{attribute 'monitoring':='call'}
//List of movers managed by this station
PROPERTY AssignedMovers : I_CH_List
GET
AssignedMovers := THIS^.fbAssignedMovers;
END_GET
END_PROPERTY

METHOD DeleteMoversQueue : HRESULT
VAR
	ipTempMover : I_XP_Mover;
END_VAR
//Not allowed in enabled state
IF THIS^.ipXPSystem.Enabled THEN
	DeleteMoversQueue := E_FAIL;
	RETURN;
END_IF


//Delete intormation in linked mover
THIS^.fbAssignedMovers.ResetIterator();
WHILE THIS^.fbAssignedMovers.HasNextObject() DO
	IF ToXPMover(THIS^.fbAssignedMovers.GetNextObject(),ipTempMover) THEN
		ipTempMover.ParentStation := 0;
	END_IF	
END_WHILE

//Clear list
fbAssignedMovers.Clear();

DeleteMoversQueue := S_OK;
END_METHOD

METHOD FB_exit : BOOL
VAR_INPUT
	bInCopyCode : BOOL; // if TRUE, the exit method is called for exiting an instance that is copied afterwards (online change).
END_VAR
VAR
	pFbPath : POINTER TO FB_XP_Path;
	ipObject : I_CH_Object;
	ipPath : I_XP_Path;
END_VAR
//Clear list, delete dynamic_creation path objects
WHILE NOT THIS^.fbListPathAhead.IsEmpty DO
	ipObject := fbListPathAhead.GetRandomObject();
	fbListPathAhead.RemoveObject(ipObject);
	
	__QUERYINTERFACE(ipObject, ipPath) ;
	pFbPath := ipPath.PointerToThis;
	__DELETE(pFbPath);
END_WHILE
END_METHOD

METHOD FB_init : BOOL
VAR_INPUT
	bInitRetains : BOOL; // if TRUE, the retain variables are initialized (warm start / cold start)
	bInCopyCode : BOOL;  // if TRUE, the instance afterwards gets moved into the copy code (online change)
	
	ipSystem 			: I_CH_Object;
	ipAccocietedTrack 	: I_XP_Track;//track on which the station is located
	sUniqueName			: STRING;		//expl.:'Loading' unique identification for this station
	sTargetGroup		: STRING;	//to which group of stations does this station belong? e.g. several stations can belong to one 'Infeed' if this is implemented redundantly.
	nMoverQueueSize 	: UINT;
	xPos				: LREAL; 	
	yPos				: LREAL; 	
END_VAR

VAR_INST
	{attribute 'hide'}
	bFBInitCalledOnce : BOOL; //Do the following code once during start up and not during onlinechange
END_VAR

VAR 



END_VAR
//Do the following code once during start up and not during onlinechange
IF NOT bFBInitCalledOnce THEN 
	
	(* Register to the Xplanar System
	   1. Test if the interface exists
	   2. Test if the object implements a "System for Mover" interface 
	*)
	IF ipSystem <> 0 AND_THEN __QUERYINTERFACE(ipSystem,THIS^.ipXpSystem) THEN
		THIS^.ipXpSystem.RegisterStation(THIS^);
	ELSE
		bErrorDuringFbInit := TRUE;
	END_IF

	
	// 0 = get closest track (in step configure)
	IF ipAccocietedTrack <> 0 THEN
		THIS^.ipAccocietedTrack := ipAccocietedTrack;
		bTrackIsSetInFbInit := TRUE;
	END_IF
	 
	
	//"" is maybe entered in an waiting or dynamic station and the name is not important
	IF sUniqueName <> '' THEN 
		THIS^.fbSourceInfo.sName := sUniqueName;
	ELSE
		sUniqueName := THIS^.fbSourceInfo.sName;
	END_IF

	
	//"" is maybe entered in an waiting or dynamic station and the name is not important
	IF sTargetGroup <> '' THEN 
		THIS^.sTargetGroup := sTargetGroup;
	ELSE
		THIS^.sTargetGroup := THIS^.fbSourceInfo.sName;
	END_IF

	
	THIS^.nMoverQueueSize 		:= nMoverQueueSize;
	THIS^.fbPositionPlanned.x 	:= xPos;
	THIS^.fbPositionPlanned.y 	:= yPos;


	THIS^.fbTrigger.FB_init(FALSE,FALSE, THIS^.ipXpSystem);

END_IF

bFBInitCalledOnce := TRUE;
END_METHOD

{attribute 'monitoring':='call'}
PROPERTY Feedback : I_CH_Feedback
GET
Feedback := THIS^.fbFeedback;
END_GET
END_PROPERTY

{attribute 'monitoring':='call'}
//Filter content, movers with one of these targets may not approach or drive over the station
PROPERTY Filter : STRING
GET
Filter := sFilter;
END_GET
SET
sFilter := Filter;
END_SET
END_PROPERTY

(*THIS METHOD uses the A* algorithm TO find the shortest route TO the destination in the network. Returns an INTERFACE with information about the destination found, such as station, path TO destination, path length.
If an interface=0 is returned, then no path can be found at the current time.*)
METHOD GetPathToTarged : I_PathAStarNode
VAR_INPUT
	sTargedStation : REFERENCE TO STRING; //unique station name or group of stations. EmptyString=Any
END_VAR
VAR	
	nDifZero : INT;	///zzz remove

	nIdx : UDINT;
	bCorrectLUID: BOOL;
	bCorrectGroupe : BOOL;
	bFilterBlockThisMover : BOOL;
	bStationIsBlocked : BOOL;
	bDummyStation : BOOL; //Station without movers only to change the dynamics of passing movers;
	bTargedFound : BOOL;
	bImTheAsker : BOOL; // Do not return this station as a targed

	ipActiveStationAStar : I_PathAStarNode;
	ipEmptyPathObj : I_PathAStarNode;
	ipEachPathAhead : I_XP_Path;
	ipPathFoundInOpenList : I_PathAStarNode;
	ipEachAStarNode : I_PathAStarNode;
	ipBesStationAStar : I_PathAStarNode;	
	ipThisStation : I_XP_Station := THIS^;
	
	fPathLength : LREAL;
END_VAR
VAR_INST
	fbLastFoundResult : FB_AStarNode;
END_VAR
VAR_STAT
	fbListNotUsedNodes : FB_CH_List; // Use GetNext() to allways get a not used one
	afbPathAStarNodes : ARRAY[0..(CHALET_BaseComponents.BaseParameterlist.MAX_OBJECTS-1)] OF FB_AStarNode;	
	fbListOpen : FB_CH_List; //To check
	fbListClosed : FB_CH_List; //Allready checked	
END_VAR
//only on first call, add nodes to list of not used objects
IF fbListNotUsedNodes.IsEmpty THEN
	FOR nIdx := 0 TO (CHALET_BaseComponents.BaseParameterlist.MAX_OBJECTS-1) DO
		fbListNotUsedNodes.AddObject(afbPathAStarNodes[nIdx]);
	END_FOR
END_IF

//Clear list
fbListOpen.Clear();
fbListClosed.Clear();

//Init objects in list
fbListNotUsedNodes.ResetIterator();
WHILE fbListNotUsedNodes.HasNextObject() DO
	IF __QUERYINTERFACE(fbListNotUsedNodes.GetNextObject(), ipEachAStarNode) THEN
		IF 	ipEachAStarNode.Station = 0 THEN
			EXIT;//Last used element found, abort
		END_IF
	
		ipEachAStarNode.Station := 0;
		ipEachAStarNode.RouteUsedToNode.Clear();
	END_IF
END_WHILE

//Reset last found result
fbLastFoundResult.Station := 0;
fbLastFoundResult.RouteUsedToNode.Clear();

// Reset once - Use GetNext() to allways get a not used one
fbListNotUsedNodes.ResetIterator();

//This is the start of the search operation. Add this station
__QUERYINTERFACE(fbListNotUsedNodes.GetNextObject(), ipEmptyPathObj);
ipEmptyPathObj.Station := (THIS^);
fbListOpen.AddObject(ipEmptyPathObj);

WHILE NOT fbListOpen.IsEmpty DO
	//Get objet from list with smallest distanse to start-station

	__QUERYINTERFACE(fbListOpen.GetObjectWithLowestNumber(), ipActiveStationAStar);
	//Move objet from open to closed list
	fbListOpen.RemoveObject(ipActiveStationAStar);
	fbListClosed.AddObject(ipActiveStationAStar);
	
	IF ipActiveStationAStar = 0 THEN
		//zzz todo error, this should never happen
		nDifZero := nDifZero / nDifZero;
		CONTINUE;
	END_IF
	
	IF ipBesStationAStar <> 0 AND_THEN ipActiveStationAStar.PathLength > ipBesStationAStar.PathLength THEN
		// if a valid station is allreadyx known, skip all station who allready have a larger distance
		CONTINUE;
	END_IF
	
	bImTheAsker := ipActiveStationAStar.Station = ipThisStation;
	bCorrectLUID := (ipActiveStationAStar.Station.LUID = sTargedStation);
 	bCorrectGroupe := (ipActiveStationAStar.Station.TargetGroupe = sTargedStation) OR (sTargedStation =  XPlanarParameterlist.S_ANY_STATION_NAME);
	bDummyStation := (ipActiveStationAStar.Station.MoverQueueSize = 0);//Station without movers only to change the dynamics of passing movers;
	bFilterBlockThisMover := (ipActiveStationAStar.Station.Filter <>  XPlanarParameterlist.S_ANY_STATION_NAME) AND (ipActiveStationAStar.Station.Filter <> sTargedStation) AND NOT bCorrectLUID; // Correct LUID is stronger than filter
	bStationIsBlocked := (ipActiveStationAStar.Station.CtsEmptySpaceInQueue <= 0 AND NOT bDummyStation) OR NOT ipActiveStationAStar.Station.ReadyToRecvMovers;

	IF (bFilterBlockThisMover OR bStationIsBlocked) AND NOT bImTheAsker THEN
		//Skip
		CONTINUE;
	END_IF
	
	
	IF (bCorrectLUID OR bCorrectGroupe) AND NOT bImTheAsker AND NOT bDummyStation THEN
		//FOUND! - check if way is shorter
		IF ipBesStationAStar=0 OR_ELSE  ipActiveStationAStar.PathLength <= ipBesStationAStar.PathLength THEN
			//shorter - store
			ipBesStationAStar := ipActiveStationAStar;
		END_IF
		
	ELSE		
		// If the destination has not yet been found, set the successor nodes of the current node to the open list
		ipActiveStationAStar.Station.PathsAhead.ResetIterator();
		WHILE ipActiveStationAStar.Station.PathsAhead.HasNextObject() DO
			__QUERYINTERFACE(ipActiveStationAStar.Station.PathsAhead.GetNextObject(), ipEachPathAhead); 
			
			IF fbListClosed.LUIDInList(ipEachPathAhead.StationDestination.LUID) THEN
				// if the successor node is already on the closed list - do nothing, repeate WHILE loop
				CONTINUE;
			END_IF
			
			//Calculate distance to start oh the new found station
			fPathLength := ipActiveStationAStar.PathLength + ipEachPathAhead.Length;
		
			//Check if this station is allready existin in open list - compare if this one is shorter
			IF __QUERYINTERFACE( fbListOpen.FindLUID(ipEachPathAhead.StationDestination.LUID), ipPathFoundInOpenList)  THEN
				IF ipPathFoundInOpenList.PathLength <= fPathLength  THEN
					//object in open list is shorter - do nothing, repeate WHILE loop
					CONTINUE;
				ELSE
					//new object is shorter - remove old object in open lsit
					fbListOpen.RemoveObject(ipPathFoundInOpenList);
				END_IF
			END_IF			
			
			
			//Add this path ahead to open list - set new length
			__QUERYINTERFACE(fbListNotUsedNodes.GetNextObject(), ipEmptyPathObj);
			ipEmptyPathObj.Station := ipEachPathAhead.StationDestination;
			ipEmptyPathObj.RouteUsedToNode.Duplicate(ipActiveStationAStar.RouteUsedToNode);
			ipEmptyPathObj.RouteUsedToNode.AddObject(ipEachPathAhead);
			fbListOpen.AddObject(ipEmptyPathObj);

		END_WHILE
		ipActiveStationAStar.Station.PathsAhead.RestoreIterator();

	END_IF

END_WHILE


//Return station or nothing
IF ipBesStationAStar = 0 THEN
	GetPathToTarged := 0;
ELSE
	//store list in an instance
	fbLastFoundResult.Station := ipBesStationAStar.Station;
	fbLastFoundResult.RouteUsedToNode.Duplicate(ipBesStationAStar.RouteUsedToNode);
	GetPathToTarged := fbLastFoundResult;
END_IF
END_METHOD

METHOD Initialize : HRESULT
VAR
	ipEachStationAhead : I_XP_Station;
	nIdx : UDINT;
END_VAR
VAR_INST
	//This error cannot be reset. Requires a reset cold
	{attribute 'hide'}	
	fbInitError : FB_TcAlarm;
	{attribute 'hide'}	
	fbMissingInterfaceAlarm : FB_TcAlarm;
END_VAR
//Check Error during FB_Init
IF THIS^.bErrorDuringFbInit THEN
	IF NOT fbInitError.bRaised THEN 
		//This error cannot be reset. Requires a reset cold
		fbInitError.CreateEx(stEventEntry:=TC_EVENTS.CHALET_Base_Events.ErrorFBinit, ipSourceInfo := THIS^.fbSourceInfo, bWithConfirmation := FALSE);
		fbInitError.Raise(0);
	END_IF
	Initialize:= E_FAIL;
	THIS^.fbFeedback.HR := Initialize;
	RETURN;
END_IF	

//Interface to System is missing
IF THIS^.ipXpSystem = 0 THEN
	IF NOT fbMissingInterfaceAlarm.bRaised THEN 
		//This error cannot be reset. Requires a reset cold
		fbMissingInterfaceAlarm.CreateEx(stEventEntry:=TC_EVENTS.CHALET_Base_Events.ErrorFBinit, ipSourceInfo := THIS^.fbSourceInfo, bWithConfirmation := FALSE);
		fbMissingInterfaceAlarm.Raise(0);
	END_IF
	Initialize := E_FAIL;
	THIS^.fbFeedback.HR := Initialize;
	RETURN;
END_IF


IF NOT THIS^.bInitDone THEN
	//Busy
	Initialize:= S_PENDING;
	
	//Clean up
	THIS^.DeleteMoversQueue();


	bInitDone := TRUE;
ELSE
	//Done
	Initialize:= S_OK;
END_IF


THIS^.fbFeedback.ActiveCommand 		:= TO_STRING(CHALET_NC.E_NcAxisCommands.Initialize);
THIS^.eActiveCommand 				:= CHALET_NC.E_NcAxisCommands.Initialize;
THIS^.fbFeedback.LastCommandAccepted:= TRUE;	
//Set done or keep in busy state	
THIS^.fbFeedback.HR := Initialize;
END_METHOD

{attribute 'monitoring':='call'}
//[mm] Every mover that leaves or passes the station gets this new gap as a target.
PROPERTY MoverGapAtExit : LREAL
GET
MoverGapAtExit := fMoverGapAtExit;
END_GET
SET
IF MoverGapAtExit < XPlanarParameterlist.F_MOVER_MINIMUM_GAP_ON_TRACK THEN
	MoverGapAtExit := XPlanarParameterlist.F_MOVER_MINIMUM_GAP_ON_TRACK;
END_IF

fMoverGapAtExit := MoverGapAtExit;
END_SET
END_PROPERTY

{attribute 'monitoring':='call'}
//Unique object ID
PROPERTY OID : OTCID
GET
OID := THIS^.fbOptionalTrackUsedInLiveView.MCTOPLC_STD.TrackOID;
END_GET
END_PROPERTY

{attribute 'monitoring':='call'}
//List of paths that lead to stations before this station
PROPERTY PathsAhead : I_CH_List
GET
PathsAhead := THIS^.fbListPathAhead;
END_GET
END_PROPERTY

{attribute 'monitoring':='call'}
//List of paths that lead to stations behind this station
PROPERTY PathsBehinde : I_CH_List
GET
PathsBehinde := THIS^.fbListPathBehind;
END_GET
END_PROPERTY

{attribute 'monitoring':='call'}
//[mm] from the beginning of the assigned track
PROPERTY PositionOnTrack : LREAL
GET
PositionOnTrack := THIS^.fPositionOnTrack;
END_GET
END_PROPERTY

{attribute 'monitoring':='call'}
//Position on the assigned track
PROPERTY PositionOnTrackXY : REFERENCE TO PositionXY
GET
PositionOnTrackXY REF= THIS^.fbPositionOnTrackXY;
END_GET
END_PROPERTY

{attribute 'monitoring':='call'}
//Planned position, not necessarily on the track. Only changeable when the system is disabled
PROPERTY PositionXY : REFERENCE TO  PositionXY
GET
PositionXY REF= THIS^.fbPositionPlanned;
END_GET
END_PROPERTY

(* 
	Use this Methode to calculate time sensitive date once each cycle. Example: read analog input and convert before do get Signal propertie
*)
METHOD PROTECTED Prepare : HRESULT
VAR_INST
	{attribute 'hide'}	
	nLastUpdatedCycleCount : UDINT;
END_VAR

VAR
	nLoopIndex : UINT;
	fExpectedDistanceToParent : LREAL;
	nCycleTime_ms : UDINT;
	bMoverInQueue : BOOL;
	bTempMoverInPosition : BOOL;
	bTempMoverVeloZero : BOOL;
	bTempMoverInMonitoringTime : BOOL;
	bTempMoverThisStationAsTarged : BOOL;
END_VAR
VAR_INST
	{attribute 'hide'}
	nCycleCountInPos : UDINT;
END_VAR
//Check if this Cycle the dates are allready prepared. This is important for time sensitive informations.
IF nLastUpdatedCycleCount <> TwinCAT_SystemInfoVarList._TaskInfo[THIS^.TaskIndex].CycleCount THEN
	nLastUpdatedCycleCount := TwinCAT_SystemInfoVarList._TaskInfo[THIS^.TaskIndex].CycleCount ;


	(* Check if mover is in place. Time and Position window *)
	//If queuesize is zero, mover is never in place.
	IF nMoverQueueSize = 0 OR THIS^.ipAccocietedTrack = 0 OR NOT ipXpSystem.Enabled THEN
		THIS^.bMoversInPlace := FALSE;
		nCycleCountInPos := 0;
	ELSE
		//Get this task cycle Count and time 
		nCycleTime_ms := TwinCAT_SystemInfoVarList._TaskInfo[THIS^.nTaskIndex].CycleTime(*100ns*) / 10_000 ;
		
		bTempMoverInPosition := TRUE; bTempMoverVeloZero := TRUE; bTempMoverThisStationAsTarged := TRUE;
		fExpectedDistanceToParent := 0;
		FOR nLoopIndex := 0 TO (THIS^.nMoverQueueSize-1) DO
			IF THIS^.fbSortedListMoversInQueue.MoversInZone[nLoopIndex] <> 0 THEN
				//Check position and Gap - 1 mover do not have a gap
				IF nLoopIndex <> 0 THEN
					fExpectedDistanceToParent := fExpectedDistanceToParent + THIS^.fbSortedListMoversInQueue.MoversInZone[nLoopIndex].LastCmdTargedGap;
				END_IF
				bMoverInQueue		:= TRUE;
				bTempMoverInPosition := bTempMoverInPosition AND (ABS(THIS^.fbSortedListMoversInQueue.MoversInZone[nLoopIndex].DistToParentStation - fExpectedDistanceToParent) <= fTargetPosWindow );
				bTempMoverVeloZero := bTempMoverVeloZero AND (THIS^.fbSortedListMoversInQueue.MoversInZone[nLoopIndex].PlanarMover.MCTOPLC.SETONTRACK.SetVelo = 0.0);
				bTempMoverThisStationAsTarged := bTempMoverThisStationAsTarged AND ((THIS^.fbSortedListMoversInQueue.MoversInZone[nLoopIndex].TargetStation = THIS^.TargetGroupe) OR (THIS^.fbSortedListMoversInQueue.MoversInZone[nLoopIndex].TargetStation = THIS^.LUID));
			ELSE
				//Missing mover in queue
				bMoverInQueue := FALSE;
				EXIT;
			END_IF
		END_FOR
			
		//start time if mover position is ok
		IF bTempMoverInPosition  THEN
			nCycleCountInPos := nCycleCountInPos + 1;
		ELSE
			nCycleCountInPos := 0;
		END_IF
		
		bTempMoverInMonitoringTime := (UDINT_TO_TIME(nCycleCountInPos * nCycleTime_ms) >= tTargetPosMonitoringTime);
				
		THIS^.bMoversInPlace := bMoverInQueue AND bTempMoverInPosition AND bTempMoverInMonitoringTime AND bTempMoverThisStationAsTarged;// AND bTempMoverVeloZero;
	END_IF
	
	
END_IF
END_METHOD

{attribute 'monitoring':='call'}
//List of stations before this station
PROPERTY StationsAhead : I_CH_List
GET
StationsAhead := THIS^.fbStationsAhead;
END_GET
END_PROPERTY

{attribute 'monitoring':='call'}
//List of stations behinde this station
PROPERTY StationsBehinde : I_CH_List
GET
StationsBehinde := THIS^.fbStationsBehinde;
END_GET
END_PROPERTY

METHOD Update : HRESULT
VAR
	iStation: I_XP_Station;
	bValideStationToStartMove : BOOL;
	ipThisStation : I_XP_Station := THIS^;
	ipPath : I_XP_Path;
	ipRoute : I_CH_List;
	ipMover : I_XP_Mover;
	bValideInterface, bMoverOnSameTrack, bInDecisionDistance : BOOL;
	nIdx : UDINT;
	bStationIsBlocked : BOOL;
END_VAR
//Force to do init befor call update
IF NOT bInitDone THEN
	THIS^.Initialize();
	RETURN;
END_IF

THIS^.Prepare();//Prepare time-critical information, if not already done


// ********************** Set feedback depending on active command *******************************
IF THIS^.eActiveCommand <> E_NcAxisCommands.None THEN
	fbFeedback.ActiveCommand 	:= TO_STRING(THIS^.eActiveCommand);	
END_IF

CASE THIS^.eActiveCommand OF

	E_NcAxisCommands.Initialize:
		fbFeedback.Busy 			:= NOT THIS^.bInitDone;
		fbFeedback.Done 			:= THIS^.bInitDone;
		fbFeedback.ErrorId 			:= 0;
		                        	

	ELSE//External command in subclass
		;
END_CASE


// **********************  Stop to execute commands on .done or .error ***************************
IF fbFeedback.Done OR THIS^.fbFeedback.Error THEN
	eActiveCommand 				:= E_NcAxisCommands.None;
END_IF



// **********************  OnMoverPasses ***************************
// Detect mover who is passing the station and call method for easier overwriting
IF fbTrigger.MoverDetected AND (fbTrigger.MoverAtTrigger <> 0) THEN
	THIS^.OnMoverPasses(fbTrigger.MoverAtTrigger);
END_IF


// **********************  If enabled start station logic ***************************
IF THIS^.ipXpSystem.Enabled THEN
	
	// Process Simulation. 	
	// All functionality packed into one method for easier overwriting
	THIS^.UpdateSimulation();
	
		
	// Interaction with the movers. Sending on to the next station. 
	// All functionality packed into one method for easier overwriting
	THIS^.UpdateMoverInteraction();
	
	
	//The movers have a list of waypoints that they have to travel to on the way to the destination station. 
	//It is checked whether this station is one of these waypoints
	// - if yes, send the mover to the next waypoint and remove this stop from the list
	//Do not wait until mover is at station possition, use fDecisionDistance
	ipXpSystem.Movers.ResetIterator();
	WHILE ipXpSystem.Movers.HasNextObject() DO
		IF __QUERYINTERFACE(ipXpSystem.Movers.GetNextObject(),ipMover) THEN
			ipRoute := ipMover.Route;
			bValideInterface 	:= ipRoute <> 0;
			bMoverOnSameTrack 	:= ipMover.CurrentTrack = ipThisStation.AccocietedTrack;
			bInDecisionDistance := (ABS(ipMover.PositionOnTrack - ipThisStation.PositionOnTrack) < THIS^.fDecisionDistance);
		ELSE 
			bValideInterface := FALSE; bMoverOnSameTrack := FALSE; bInDecisionDistance := FALSE;
		END_IF		
		
		IF bValideInterface AND bMoverOnSameTrack AND bInDecisionDistance THEN
			ipRoute.ResetIterator();
			WHILE ipRoute.HasNextObject() DO
				IF __QUERYINTERFACE(ipRoute.GetNextObject(), ipPath) AND_THEN ipPath.StationStart = ipThisStation THEN
					//Remove this path from route and send to path desination
					ipMover.Route.RemoveObject(ipPath);
					
					//Set new dynamic. Be careful when reducing the deceleration so that the mover can still stop in real time
					IF XPlanarParameterlist.B_STATIONS_OVERRIDE_MOVER_DYN_CONSTRAINT THEN
						ipMover.SetDynConstraint_Path(	V:= THIS^.fMoverVeloAtExit, 
								A:= THIS^.fMoverAccAtExit,
								D:= THIS^.fMoverDecAtExit,
								J:= MC_DEFAULT);
					END_IF

					
					//If mover is standstill in current station, send him away whit the exit gap, else use the in mover stored gap
					IF (ABS(ipMover.PositionOnTrack - THIS^.PositionOnTrack) <= 1.0) THEN
						ipMover.MoveOnTrackToStation(ipStation := ipPath.StationDestination,
													fGap:= THIS^.fMoverGapAtExit);					
					ELSE
						ipMover.MoveOnTrackToStation(ipStation := ipPath.StationDestination,
													fGap:= ipMover.LastCmdTargedGap);
					END_IF	
				END_IF
			END_WHILE
			ipRoute.RestoreIterator();
		END_IF		
	END_WHILE
	ipXpSystem.Movers.RestoreIterator();
	
	
	//Check for errors
	(*The station is blocked. 
	The first mover in the row is correctly positioned in the station. 
	The queue has a size of >1, but now the n+1 mover does not have this station as its destination. 
	However, it cannot overtake. The station never gives the process a ready signal.*)
	IF THIS^.MoverQueueSize > 1 AND THIS^.MoversInQueue[0] <> 0 AND_THEN (THIS^.MoversInQueue[0].TargetStation = THIS^.TargetGroupe OR THIS^.MoversInQueue[0].TargetStation = THIS^.LUID) THEN
		FOR nIdx := 1 TO (CHALET_BaseComponents.BaseParameterlist.MAX_OBJECTS-1) DO
			//Search for Mover with a direrent targed
			IF THIS^.MoversInQueue[nIdx] <> 0 AND_THEN NOT(THIS^.MoversInQueue[nIdx].TargetStation = THIS^.TargetGroupe OR THIS^.MoversInQueue[nIdx].TargetStation = THIS^.LUID) THEN
				//Error
				bStationIsBlocked := TRUE;
				IF NOT fbAlarmStationIsBlocked.bRaised THEN
					//Station is blocked. Mover {0} has {1} as target position but cannot overtake
					fbAlarmStationIsBlocked.CreateEx(TC_Events.CHALET_XPlanar_Events.StationIsBlocked,0,THIS^.fbSourceInfo);
					fbAlarmStationIsBlocked.ipArguments.AddStringByValue(THIS^.MoversInQueue[nIdx].LUID).AddStringByValue(THIS^.MoversInQueue[nIdx].TargetStation);
					fbAlarmStationIsBlocked.Raise(0);
					EXIT;					
				END_IF
			END_IF
		END_FOR
	END_IF
	IF NOT bStationIsBlocked AND fbAlarmStationIsBlocked.bRaised THEN
		fbAlarmStationIsBlocked.Clear(0,0);
	END_IF
	
	
END_IF



// **********************  If disabled clear some bits ***************************
IF NOT THIS^.ipXpSystem.Enabled THEN
	fbAlarmStationIsBlocked.Clear(0,0);
END_IF

Update := S_OK;
END_METHOD

METHOD PROTECTED UpdateMoverInteraction : HRESULT
VAR
	ipFirstMoverInQueue: I_XP_Mover;
	sTargedStation : STRING;
	bMoverValideToSendAway : BOOL;
	bInReachForNewCmd : BOOL;
	bThisStationAsParent : BOOL;
	bFilterDoesNotAllowThisMover : BOOL;
	bThisStationAsTarged : BOOL;
	bMoverIsNotOnAWaitingStation : BOOL;
	bStationInBlockedTryToSolve : BOOL; //Send 1. Mover away ignore that already in correct station
	bMoverMustLeaveTheStation : BOOL; //Set from external
	bSearchNewDestination : BOOL;
	bStationCanBeReachedWhitoutBranch : BOOL;
	bStationIsOverfilled : BOOL;

	ipStationAhead : I_XP_Station;
	ipPathFoundAStarValide : I_PathAStarNode;
	ipPathFoundAStarAnyStation : I_PathAStarNode;
	ipRouteUsed : I_XP_Path;
	
	fbListOf : FB_AStarNode;
END_VAR
//Get first mover in this station
IF NOT __QUERYINTERFACE(THIS^.MoversInQueue[0],ipFirstMoverInQueue) THEN
	//No valide interface. (Mover not present)
	RETURN;
END_IF


//Get a few helpful variables
sTargedStation := ipFirstMoverInQueue.TargetStation;
bThisStationAsTarged := (sTargedStation = THIS^.TargetGroupe) OR (sTargedStation = THIS^.LUID); 
bThisStationAsParent := ipFirstMoverInQueue.ParentStation.LUID = THIS^.LUID;
bMoverIsNotOnAWaitingStation := NOT(bThisStationAsParent AND NOT bThisStationAsTarged AND (THIS^.MoverQueueSize > 0));
bInReachForNewCmd	:= (ipFirstMoverInQueue.DistToParentStation <= THIS^.fDecisionDistance);	
bStationInBlockedTryToSolve  := THIS^.fbAlarmStationIsBlocked.bRaised;//Send 1. Mover away ignore that already in correct station
bFilterDoesNotAllowThisMover := (THIS^.Filter <> XPlanarParameterlist.S_ANY_STATION_NAME) AND (THIS^.Filter <> sTargedStation);
bMoverMustLeaveTheStation := THIS^.nCtsMoversMustLeaveThisStation > 0;
bStationIsOverfilled  := THIS^.CtsMoversInQueue > THIS^.nMoverQueueSize;


//Decide what happens to the mover
bSearchNewDestination := bInReachForNewCmd AND bThisStationAsParent AND (NOT bThisStationAsTarged OR bMoverMustLeaveTheStation OR bStationInBlockedTryToSolve OR bStationIsOverfilled);
IF bSearchNewDestination THEN
	
	//1. Prio - Get a direct path to targed - Only if specific
	IF sTargedStation <> XPlanarParameterlist.S_ANY_STATION_NAME THEN
		ipPathFoundAStarValide := GetPathToTarged(sTargedStation := sTargedStation);
	END_IF

	
	
	//If path to targed is not valide, calculate once a path to any station
	IF ipPathFoundAStarValide = 0 THEN
		ipPathFoundAStarAnyStation := THIS^.GetPathToTarged(sTargedStation := XPlanarParameterlist.S_ANY_STATION_NAME);
	END_IF
	
	
	//2. Prio If the next possible station is on this track, without having to pass a switch, then go to this new station
	// The mover should be pushed as far forward as possible to avoid blocking the track
	IF  ipPathFoundAStarValide = 0 AND ipPathFoundAStarAnyStation <> 0  AND (THIS^.PathsAhead.Size = 1) AND THIS^.bNetworkHasTrackBranches THEN
		//
		ipPathFoundAStarAnyStation.RouteUsedToNode.ResetIterator();
		bStationCanBeReachedWhitoutBranch := TRUE;
		WHILE (ipPathFoundAStarAnyStation.RouteUsedToNode.HasNextObject() AND bStationCanBeReachedWhitoutBranch) DO
			IF __QUERYINTERFACE(ipPathFoundAStarAnyStation.RouteUsedToNode.GetNextObject(), ipRouteUsed) THEN
				bStationCanBeReachedWhitoutBranch := (ipRouteUsed.StationDestination.PathsAhead.Size = 1) OR (ipRouteUsed.StationDestination = ipPathFoundAStarAnyStation.Station); //Ignore if destination station have more than 1 paths ahead
			END_IF
		END_WHILE	
		ipPathFoundAStarAnyStation.RouteUsedToNode.RestoreIterator();
		IF bStationCanBeReachedWhitoutBranch THEN
			ipPathFoundAStarValide := ipPathFoundAStarAnyStation;
		END_IF
	END_IF

	
	//3. Prio - Send the mover to any station. (most time waitingstation)
	// - closest waitingstation to this station, if not allready on a waiting station
	// - if filter was maybe changed or the mover is not allowed in this station
	IF  ipPathFoundAStarValide = 0 AND ipPathFoundAStarAnyStation <> 0 AND (bMoverIsNotOnAWaitingStation OR bFilterDoesNotAllowThisMover OR bMoverMustLeaveTheStation OR bStationIsOverfilled) THEN
		ipPathFoundAStarValide := ipPathFoundAStarAnyStation;
	END_IF
END_IF


//Write new paths and parent-station to mover
IF ipPathFoundAStarValide <> 0 THEN 
	//Handover list of paths to mover
	ipFirstMoverInQueue.Route.Duplicate(ipPathFoundAStarValide.RouteUsedToNode);

	//Unregister from this station and register with a new parrent station
	THIS^.fbAssignedMovers.RemoveObject(ipFirstMoverInQueue);
	ipPathFoundAStarValide.Station.AddMoverToQueue(ipFirstMoverInQueue);	
	
	//Mover is now leaving the station
	IF THIS^.nCtsMoversMustLeaveThisStation > 0 THEN
		THIS^.nCtsMoversMustLeaveThisStation := THIS^.nCtsMoversMustLeaveThisStation - 1;
	END_IF
	
END_IF
END_METHOD

END_FUNCTION_BLOCK

// FUNCTIONs/F_GetDistToPosModulo
FUNCTION F_GetDistToPosModulo : LREAL //This is only working in Positiv Direktion
VAR_INPUT
	fTargedPosition : LREAL;
	fActualPosition : LREAL;
	fModulo 		: LREAL;
END_VAR

VAR

END_VAR

IF fTargedPosition < fActualPosition THEN
	fTargedPosition := fTargedPosition + fModulo;
END_IF

F_GetDistToPosModulo := fTargedPosition - fActualPosition;

END_FUNCTION

// COMPONENTs/System/FB_XP_System
{attribute 'no_explicit_call' := 'Do not call the body - Stick to OOP'}
(* XPlanar System - 1 per associated XPlanar 
	The system is the container and organizer for all subsequent XPlanar objects. All objects are registered with this system*)
FUNCTION_BLOCK FB_XP_System EXTENDS FB_CH_Object IMPLEMENTS I_XP_System_Registration, I_XP_System_PLC
VAR	
	{attribute 'hide'}
	bInitDone : BOOL;
	{attribute 'hide'}
	bErrorDuringFbInit : BOOL; // Not possible to reset
	{attribute 'hide'}                   	
	eActiveCommand 		: CHALET_Nc.E_NcAxisCommands := CHALET_Nc.E_NcAxisCommands.None;
	{attribute 'hide'}
    fbMovers     : FB_CH_List;
	{attribute 'hide'}	
    fbTracks     : FB_CH_List;
	{attribute 'hide'}	
	fbStations 	 : FB_CH_List;
	{attribute 'hide'}	
	fbTriggers 	 : FB_CH_List;
	{attribute 'hide'}	
	fbZones 	 : FB_CH_List;
	{attribute 'hide'}	
	fbPaths 	 : FB_CH_List;
	{attribute 'hide'}	
    ipGroup       : I_XP_Group;
	{attribute 'hide'}	
    ipEnvironment : I_XP_Environment;
	{attribute 'hide'}
    nSeqEnabling  : UINT;
	{attribute 'hide'}
	nSeqJoiningTrack : UINT;
	{attribute 'hide'}
	nSeqJoiningStation : UINT;
	{attribute 'hide'}	
    nSeqDisabling  : UINT := SEQ_DONE;
	{attribute 'hide'}
	fbFeedback : FB_CH_Feedback(ipSourceInfo := fbSourceInfo);	
END_VAR
VAR CONSTANT
	{attribute 'hide'}
	SEQ_DONE : UINT := 999;
END_VAR

METHOD PROTECTED JoiningStation : HRESULT
VAR
	hr : HRESULT;
	ipEachMover : I_XP_Mover;
	ipEachMoverPlc : I_XP_Mover_PLC;
	ipEachMoverInStation : I_XP_Mover;
	ipEachStation : I_XP_Station;
	ipFirstStation : I_XP_Station;
	ipParentStation : I_XP_Station;
	ipTempMoverPlc : I_XP_Mover_PLC;
	
	//during move on track
	fVelo, fAccDec	: Tc3_Mc3Definitions.MC_LREAL := Tc3_Mc3Definitions.MC_DEFAULT;
	bError : BOOL;
	bStationNotOperational : BOOL;
	bFound : BOOL;
	
	fCalcualtedGapAtMoverPosition : LREAL;
	stPositionVector : MoverVector;
	
	ipClosestStation : I_XP_Station;
	fDistToStation : LREAL := CHALET_BaseComponents.GVL_Datatypes.cMaxLreal;
END_VAR
VAR_INST
	bResetMovers : BOOL;	

	{attribute 'hide'}	
	fbDelayJoiningStation : TON;
END_VAR
CASE nSeqJoiningStation OF

	0: //Init
		fbDelayJoiningStation.IN := FALSE;
		
		IF fbStations.IsEmpty THEN
			nSeqJoiningStation := SEQ_DONE;
		ELSE
			nSeqJoiningStation := 10;
		END_IF
	


	
		
	10:	// For each Mover, Clear planed route to targed. After enabling the tracks may have change and are not longer existing.
		THIS^.fbMovers.ResetIterator();
		WHILE THIS^.fbMovers.HasNextObject() DO
			IF __QUERYINTERFACE(THIS^.fbMovers.GetNextObject(), ipEachMover) THEN
				ipEachMover.Route.Clear();
			END_IF
		END_WHILE
		THIS^.fbMovers.RestoreIterator();
		
		//Empty Mover queue in station
		THIS^.fbStations.ResetIterator();
		WHILE THIS^.fbStations.HasNextObject() DO
			IF __QUERYINTERFACE(THIS^.fbStations.GetNextObject(), ipEachStation) THEN
				ipEachStation.DeleteMoversQueue();
			END_IF
		END_WHILE
		THIS^.fbStations.RestoreIterator();
		
		nSeqJoiningStation := 20;
	
	


	
		
	20: //Set closest station as parent station(responsible to send to targed)
		THIS^.fbMovers.ResetIterator();
		WHILE THIS^.fbMovers.HasNextObject() DO
			IF __QUERYINTERFACE(THIS^.fbMovers.GetNextObject(), ipEachMover) THEN
				
				//If the mover was very close to a station, us this station as parent
				ipClosestStation := THIS^.GetStationClosestTo(ipEachMover.LastValidPositionXYZABC);
				
				//only if the system was one enabled
				IF ipClosestStation <> 0 AND ipEachMover.LastValidTrack <> 0 THEN 
					stPositionVector.x := ipClosestStation.PositionOnTrackXY.x;
					stPositionVector.y := ipClosestStation.PositionOnTrackXY.y;
					fDistToStation := F_DistXYVectors(stPositionVector, ipEachMover.LastValidPositionXYZABC);
				END_IF

				IF fDistToStation <= 5.0(*[mm]*) THEN
					ipParentStation := ipClosestStation;
				ELSE
					ipParentStation := ipEachMover.CurrentTrack.StationAhedPosition(ipEachMover.PositionOnTrack);
				END_IF
			

				//Set as new parent
				IF ipParentStation <> 0 THEN
					ipParentStation.AddMoverToQueue(ipEachMover);
				ELSE
					//Error
					bError := TRUE;
				END_IF
			END_IF
		END_WHILE
		THIS^.fbMovers.RestoreIterator();	
	
		IF bError THEN
			nSeqJoiningStation := nSeqJoiningStation + 1000;
		ELSE
			nSeqJoiningStation := 30;	
		END_IF
	
	
	
	30: //Send Movers to targed	
		THIS^.fbMovers.ResetIterator();
		WHILE THIS^.fbMovers.HasNextObject() DO
			//Do for all Movers whitout a targed station
			IF ToXpMover(THIS^.fbMovers.GetNextObject(),ipEachMover) AND_THEN (ipEachMover.ParentStation <> 0) AND_THEN __QUERYINTERFACE(ipEachMover,ipEachMoverPlc) THEN
				//Set Path dynamic constraint to settings in XPlanarParameterlist. 0=Defalt
				IF XPlanarParameterlist.F_ENABLING_ON_TRACK_VELOCITY <> 0 THEN fVelo := XPlanarParameterlist.F_ENABLING_ON_TRACK_VELOCITY;END_IF
				IF XPlanarParameterlist.F_ENABLING_ON_TRACK_ACC_DEC <> 0 THEN fAccDec := XPlanarParameterlist.F_ENABLING_ON_TRACK_ACC_DEC;END_IF
			
				//Increase or decrease the mover DynConstraint for approaching the station 
				ipEachMoverPlc.SetDynConstraint_Path(	V:= fVelo, 
														A:= fAccDec, 
														D:= fAccDec, 
														J:= Tc3_Mc3Definitions.MC_DEFAULT);
		
				// gap depending on current position
				fCalcualtedGapAtMoverPosition := ipEachMover.CurrentTrack.GapAtPosition(ipEachMover.PositionOnTrack);
		
				hr := GetMostSignificant(hr, ipEachMover.MoveOnTrack_ShortestWay(ipTrack := ipEachMover.ParentStation.AccocietedTrack,
																				fPosition := ipEachMover.ParentStation.PositionOnTrack, 
																				fGap := fCalcualtedGapAtMoverPosition));
				
					
				END_IF
		END_WHILE
		THIS^.fbMovers.RestoreIterator();		



		IF CheckOk(hr) THEN 
			nSeqJoiningStation := 100;
		ELSIF FAILED(hr) THEN
			nSeqJoiningStation := 1000 + nSeqJoiningStation;
		END_IF	
	
	
	//	//send mover to last known targed
	//	THIS^.fbMovers.ResetIterator();
	//	WHILE THIS^.fbMovers.HasNextObject() DO
	//		IF ToXpMover(THIS^.fbMovers.GetNextObject(),ipEachMover) AND_THEN (ipEachMover.LastCmdTargedTrack <> 0) THEN
	//					hr := GetMostSignificant(hr, ipEachMover.MoveOnTrack_ShortestWay(	ipTrack		:= ipEachMover.LastCmdTargedTrack, 
	//																					  	fPosition	:= ipEachMover.LastCmdTargedPosition,
	//																					  	fGap 		:= ipEachMover.LastCmdTargedGap));
	//		END_IF
	//	END_WHILE 
	//	THIS^.fbMovers.RestoreIterator();     
	//	nSeqJoiningStation := 20;


		
	//20:	//Test if there is an Mover whitout an active parent station (first startup)
	//	//Send them to first station
	//	THIS^.fbStations.ResetIterator();
	//	IF THIS^.fbStations.HasNextObject() THEN
	//		//Get interface to first Station in list
	//		ToXpStation(THIS^.fbStations.GetNextObject(),ipFirstStation);
	//		//Set as targed station the first station in list. but as the parent the station in front of the first one(if existing) 
	//		//(the parent station is not necessarily the target station. But the station that is responsible for sending the mover forward if necessary)
	//		ipFirstStation.StationsAhead.ResetIterator();
	//		ToXpStation(ipFirstStation.StationsAhead.GetNextObject(),ipParentStation);
	//		
	//		//Check for mover whitout a targed station
	//		THIS^.fbMovers.ResetIterator();
	//		WHILE THIS^.fbMovers.HasNextObject() DO
	//			//Do for all Movers whitout a targed station
	//			IF ToXpMover(THIS^.fbMovers.GetNextObject(),ipEachMover) AND_THEN (ipEachMover.ParentStation = 0) AND_THEN __QUERYINTERFACE(ipEachMover,ipEachMoverPlc) THEN
	//				//Set Path dynamic constraint to settings in XPlanarParameterlist. 0=Defalt
	//				IF XPlanarParameterlist.F_ENABLING_ON_TRACK_VELOCITY <> 0 THEN fVelo := XPlanarParameterlist.F_ENABLING_ON_TRACK_VELOCITY;END_IF
	//				IF XPlanarParameterlist.F_ENABLING_ON_TRACK_ACC_DEC <> 0 THEN fAccDec := XPlanarParameterlist.F_ENABLING_ON_TRACK_ACC_DEC;END_IF
	//			
	//				//Increase or decrease the mover DynConstraint for approaching the station 
	//				ipEachMoverPlc.SetDynConstraint_Path(	V:= fVelo, 
	//														A:= fAccDec, 
	//														D:= fAccDec, 
	//														J:= Tc3_Mc3Definitions.MC_DEFAULT);
	//	
	//				// gap depending o current position
	//				fCalcualtedGapAtMoverPosition := ipEachMover.CurrentTrack.GapAtPosition(ipEachMover.PositionOnTrack);
	//		
	//				//Set as targed station the first station in list. but as the parent the station in front of the first one(if existing) 
	//				IF ipParentStation <> 0 THEN
	//					hr := GetMostSignificant(hr, ipEachMover.MoveOnTrackToStation(ipParentStation, fCalcualtedGapAtMoverPosition));
	//					hr := GetMostSignificant(hr, ipParentStation.AddMoverToQueue(ipEachMover));
	//				ELSE
	//					//If no partent station is existing
	//					hr := GetMostSignificant(hr, ipEachMover.MoveOnTrackToStation(ipFirstStation, fCalcualtedGapAtMoverPosition));
	//					hr := GetMostSignificant(hr, ipFirstStation.AddMoverToQueue(ipEachMover));
	//				END_IF
	//				
	//				//Only override targed if empty
	//				IF ipEachMover.TargetStation = '' THEN
	//					ipEachMover.TargetStation := ipFirstStation.TargetGroupe;
	//				END_IF
	//				
	//				
	//				//Set Path dynamic constraint back to default
	//				ipEachMoverPlc.SetDynConstraint_Path(	V:= Tc3_Mc3Definitions.MC_DEFAULT, 
	//														A:= Tc3_Mc3Definitions.MC_DEFAULT, 
	//														D:= Tc3_Mc3Definitions.MC_DEFAULT, 
	//														J:= Tc3_Mc3Definitions.MC_DEFAULT);
	//	
	//			END_IF
	//		END_WHILE 
	//		THIS^.fbMovers.RestoreIterator();
	//	END_IF
	//	
	//	IF ipParentStation <> 0 THEN
	//		//All Mover must leave this station
	//		ipParentStation.PushMoversOutOfStation();
	//	END_IF
    //
	//	nSeqJoiningStation := 30;
		
	100: //Delay to allow the movers to start movement
		fbDelayJoiningStation.IN := TRUE;
		fbDelayJoiningStation.PT := T#2S;
		IF fbDelayJoiningStation.Q THEN
			nSeqJoiningStation := 110;
			fbDelayJoiningStation.IN := FALSE;
		END_IF
	
	
	110: //Wait for all movers until the movement is completed(speed =0)
		THIS^.fbMovers.ResetIterator();
		WHILE THIS^.fbMovers.HasNextObject() DO
			IF ToXpMover(THIS^.fbMovers.GetNextObject(),ipEachMover) THEN
				//Check all movers if an error is active
				IF ipEachMover.Feedback.Error THEN
					hr := GetMostSignificant(hr, ipEachMover.Feedback.HR);
				//Wait for all movers to stop/finish movement
				ELSIF NOT (ipEachMover.Standstill) THEN
					hr := GetMostSignificant(hr, S_PENDING);
				END_IF
			END_IF
		END_WHILE 
		THIS^.fbMovers.RestoreIterator();
		
		IF CheckOk(hr) THEN 
			nSeqJoiningStation := SEQ_DONE;
		ELSIF FAILED(hr) THEN
			nSeqJoiningStation := 1000 + nSeqJoiningStation;
		END_IF			

		
	//50: // Check if a mover passes his parent station and is not abel to drive backwarts due to CA
	//	THIS^.fbMovers.ResetIterator();
	//	WHILE THIS^.fbMovers.HasNextObject() DO
	//		IF ToXpMover(THIS^.fbMovers.GetNextObject(),ipEachMover) THEN
	//			bStationNotOperational := ipEachMover.ParentStation <> 0 AND_THEN NOT ipEachMover.ParentStation.MoversInPlace;
	//			IF ipEachMover.DistToParentStation < 0 AND bStationNotOperational THEN
	//				bFound := TRUE;
	//			END_IF
	//		END_IF
	//	END_WHILE 
	//	THIS^.fbMovers.RestoreIterator();
	//	
	//	// IF found, reset all mover
	//	IF bFound OR bResetMovers THEN
	//		bResetMovers := FALSE;
	//		//Clear Mover
	//		THIS^.fbMovers.ResetIterator();
	//		WHILE THIS^.fbMovers.HasNextObject() DO
	//			IF ToXpMover(THIS^.fbMovers.GetNextObject(),ipEachMover) THEN
	//				//ipEachMover.TargetStation := '';
	//				ipEachMover.ParentStation := 0;
	//				ipEachMover.Route.Clear();
	//			END_IF
	//		END_WHILE 
	//		THIS^.fbMovers.RestoreIterator();
	//		//Clear Station
	//		THIS^.fbStations.ResetIterator();    
	//		WHILE THIS^.fbStations.HasNextObject() DO
	//			ToXpStation(THIS^.fbStations.GetNextObject(),ipEachStation);
	//			ipEachStation.DeleteMoversQueue();
	//		END_WHILE    
	//		THIS^.fbStations.RestoreIterator();   
	//		nSeqJoiningStation := 0;
	//	ELSE
	//		nSeqJoiningStation := SEQ_DONE;
	//	END_IF

	SEQ_DONE:
		;
	
	1000..1999://Error
		hr := GetMostSignificant(hr, E_FAIL);
END_CASE

//Update
fbDelayJoiningStation();


//Return value
IF FAILED(hr) THEN 
	//Error
    JoiningStation := GetMostSignificant(hr, E_FAIL);
ELSIF (nSeqJoiningStation = SEQ_DONE) THEN
	//Done
    JoiningStation := S_OK;
ELSE
	//Busy
    JoiningStation := S_PENDING;;
END_IF
END_METHOD

METHOD PROTECTED JoiningTrack : HRESULT
VAR	
	hr : HRESULT;
	ipClosestTrack, ipLastTrack : I_XP_Track;	
	ipEachMover : I_XP_Mover;
	ipEachTrack : I_XP_Track;
	fDistance : LREAL;
	fShortestDistance : LREAL;
	fDistToLastValidPos : LREAL;
	bUseClosestTrack : BOOL;
END_VAR
CASE nSeqJoiningTrack OF

	0: //Init
		IF fbTracks.IsEmpty THEN
			nSeqJoiningTrack := SEQ_DONE;
		ELSE
			nSeqJoiningTrack := 10;
		END_IF

		
	10: //Last or Closest Track	
		//compare to the last valid position whether the mover is still unchanged on the tile. 
		//If there is only a small movement <5mm, an attempt is made to move to the last position. 
		//Otherwise the closest track is moved to
		THIS^.fbMovers.ResetIterator();
		WHILE THIS^.fbMovers.HasNextObject() DO
			IF ToXpMover(THIS^.fbMovers.GetNextObject(),ipEachMover) THEN
				//Calculate distance
				fDistToLastValidPos := F_DistXYVectors(ipEachMover.LastValidPositionXYZABC, ipEachMover.PositionSet);
	
				IF fDistToLastValidPos > 5.0 OR ipEachMover.LastValidTrack = 0 THEN
					bUseClosestTrack := TRUE;
					EXIT;
				END_IF
	
			END_IF
		END_WHILE
		THIS^.fbMovers.RestoreIterator();	
		
		
		IF bUseClosestTrack THEN
			//Closest
			nSeqJoiningTrack := 50;
		ELSE
			//Last
			nSeqJoiningTrack := 60;
		END_IF
		
		
		
	50:// Join closest track
		THIS^.fbMovers.ResetIterator();
		WHILE THIS^.fbMovers.HasNextObject() DO
			IF ToXpMover(THIS^.fbMovers.GetNextObject(),ipEachMover) THEN
				
				//check all track to decide which is the closest
				//start with the greatest possible distance, so that each track is definitely closer
				fShortestDistance := CHALET_BaseComponents.GVL_Datatypes.cMaxLreal; 
				THIS^.fbTracks.ResetIterator();			
				WHILE THIS^.fbTracks.HasNextObject() DO
					IF ToXpTrack(THIS^.fbTracks.GetNextObject(),ipEachTrack) THEN
						fDistance := ipEachMover.DistToTrack(ipEachTrack);
						//closer track found
						IF fDistance <= fShortestDistance THEN
							ipClosestTrack := ipEachTrack;
							fShortestDistance := fDistance;
						END_IF
					END_IF
				END_WHILE
				THIS^.fbTracks.RestoreIterator();		
				

				IF ipClosestTrack <> 0 THEN
					hr := GetMostSignificant(hr, ipEachMover.JoinTrack(ipClosestTrack));
				ELSE
					hr := GetMostSignificant(hr, E_FAIL);
				END_IF
			
				
			END_IF
		END_WHILE
		THIS^.fbMovers.RestoreIterator();
		nSeqJoiningTrack := 100;		
		
		
	60:// Move to last known position
		THIS^.fbMovers.ResetIterator();
		WHILE THIS^.fbMovers.HasNextObject() DO
			IF ToXpMover(THIS^.fbMovers.GetNextObject(),ipEachMover) THEN
				hr := GetMostSignificant(hr, ipEachMover.MoveXY(ipEachMover.LastValidPositionXYZABC.x, ipEachMover.LastValidPositionXYZABC.y));
			END_IF
		END_WHILE
		THIS^.fbMovers.RestoreIterator();
		nSeqJoiningTrack := 61;		
		
	61: // Moving check feedback
		THIS^.fbMovers.ResetIterator();
		WHILE THIS^.fbMovers.HasNextObject() DO
			IF ToXpMover(THIS^.fbMovers.GetNextObject(),ipEachMover) THEN
				// Check mover errors
				hr := GetMostSignificant(hr, ipEachMover.Feedback.HR);
			END_IF
		END_WHILE
		THIS^.fbMovers.RestoreIterator();		
		
		IF CheckOk(hr) THEN 
			nSeqJoiningTrack := 62;
		ELSIF FAILED(hr) THEN
			nSeqJoiningTrack := 1000 + nSeqJoiningTrack;
		END_IF	
		
	62: //Join last valid track
		THIS^.fbMovers.ResetIterator();
		WHILE THIS^.fbMovers.HasNextObject() DO
			IF ToXpMover(THIS^.fbMovers.GetNextObject(),ipEachMover) THEN
				ipLastTrack := ipEachMover.LastValidTrack;
				hr := GetMostSignificant(hr, ipEachMover.JoinTrack(ipLastTrack));
			END_IF
		END_WHILE
		THIS^.fbMovers.RestoreIterator();
		nSeqJoiningTrack := 100;
		
		
	100: // Joining  track check feedback
		THIS^.fbMovers.ResetIterator();
		WHILE THIS^.fbMovers.HasNextObject() DO
			IF ToXpMover(THIS^.fbMovers.GetNextObject(),ipEachMover) THEN
				
				// Check mover errors
				hr := GetMostSignificant(hr, ipEachMover.Feedback.HR);
				
				//Check if Mover is on track
				IF NOT (ipEachMover.Mode = MC_PLANAR_MOVER_COMMAND_MODE.OnTrack) THEN
					hr := GetMostSignificant(hr, S_PENDING);
				END_IF
			END_IF
		END_WHILE
		THIS^.fbMovers.RestoreIterator();
		
		IF CheckOk(hr) THEN 
			nSeqJoiningTrack := SEQ_DONE;
		ELSIF FAILED(hr) THEN
			nSeqJoiningTrack := 1000 + nSeqJoiningTrack;
		END_IF			

		
	1000..1999://Error
		hr := GetMostSignificant(hr, E_FAIL);
END_CASE

		
		
//Return value
IF FAILED(hr) THEN 
	//Error
    JoiningTrack := GetMostSignificant(hr, E_FAIL);
ELSIF (nSeqJoiningTrack = SEQ_DONE) THEN
	//Done
    JoiningTrack := S_OK;
ELSE
	//Busy
    JoiningTrack := S_PENDING;;
END_IF
END_METHOD

METHOD Disable : I_CH_Feedback
VAR_INPUT
END_VAR
//Disable is allways posible, but only if not already active

IF THIS^.nSeqDisabling = 0 OR THIS^.nSeqDisabling >= SEQ_DONE THEN
	THIS^.nSeqDisabling 	:= 1;
	THIS^.nSeqEnabling 		:= 0;
	
	THIS^.eActiveCommand 					:= CHALET_NC.E_NcAxisCommands.Disable;
	THIS^.fbFeedback.LastCommandAccepted	:= TRUE;		
	THIS^.fbFeedback.Busy 					:= TRUE;
			
	
ELSE
	THIS^.fbFeedback.LastCommandAccepted	:= FALSE;	
END_IF

Disable := THIS^.fbFeedback;
END_METHOD

{attribute 'monitoring':='call'}
PROPERTY Disabled : BOOL
GET
Disabled := nSeqDisabling = SEQ_DONE OR 
			(nSeqDisabling = 0 AND nSeqEnabling = 0);
END_GET
END_PROPERTY

METHOD PROTECTED Disabling : HRESULT
VAR
	hr : HRESULT;
	bOk : BOOL := TRUE;
	iTempMover : I_XP_Mover;
	iTempTrack : I_XP_Track;
END_VAR
VAR_INST
	hrLastCycle : HRESULT;
END_VAR
Disabling := S_PENDING;
CASE nSeqDisabling OF
	0: // Idle
		Disabling := S_OK;
		
		
	1: // Halt movers - keep at first position for a fast stop reaction
		THIS^.fbMovers.ResetIterator();
		WHILE THIS^.fbMovers.HasNextObject() DO
			IF ToXpMover(THIS^.fbMovers.GetNextObject(),iTempMover) THEN
				hr := GetMostSignificant(hr, iTempMover.Halt());
			END_IF
		END_WHILE
		THIS^.fbMovers.RestoreIterator();
		
		IF CheckOk(hr) THEN 
			nSeqDisabling := 20;
		ELSE
			nSeqDisabling := 1000 + nSeqDisabling;
		END_IF	
	
		
	20: // Halting movers
		THIS^.fbMovers.ResetIterator();
		WHILE THIS^.fbMovers.HasNextObject() DO
			IF ToXpMover(THIS^.fbMovers.GetNextObject(),iTempMover) THEN
				bOk := bOk AND iTempMover.Standstill;
			END_IF
		END_WHILE
		THIS^.fbMovers.RestoreIterator();
		
		IF bOk THEN 
			nSeqDisabling := 30;
		END_IF	
			
		
	
	30: // Reset movers
		THIS^.fbMovers.ResetIterator();
		WHILE THIS^.fbMovers.HasNextObject() DO
			IF ToXpMover(THIS^.fbMovers.GetNextObject(),iTempMover) THEN
				hr := GetMostSignificant(hr, iTempMover.Reset());
			END_IF
		END_WHILE
		
		IF CheckOk(hr) THEN 
			nSeqDisabling := 40;
		ELSE
			nSeqDisabling := 1000 + nSeqDisabling;
		END_IF		
		
		
	40: // Resetting movers
		THIS^.fbMovers.ResetIterator();
		WHILE THIS^.fbMovers.HasNextObject() DO
			IF ToXpMover(THIS^.fbMovers.GetNextObject(),iTempMover) THEN
				hr := GetMostSignificant(hr, iTempMover.Feedback.HR);
			END_IF
		END_WHILE
		
		IF CheckOk(hr) THEN 
		//	nSeqDisabling := 45;
			nSeqDisabling := 50;
		ELSIF FAILED(hr) THEN
			nSeqDisabling := 1000 + nSeqDisabling;
		END_IF
		
		
		
(*		
	45: // Stop external Setpoint 
		THIS^.fbMovers.ResetIterator();
		WHILE THIS^.fbMovers.HasNextObject() DO
			IF ToXpMover(THIS^.fbMovers.GetNextObject(),iTempMover) THEN
				hr := GetMostSignificant(hr, iTempMover.StopExternalSetpoint());
			END_IF
		END_WHILE
		
		IF CheckOk(hr) THEN 
			nSeqDisabling := 46;
		ELSE
			nSeqDisabling := 1000 + nSeqDisabling;
		END_IF			
		

	46: // Stoping external Setpoint 
		THIS^.fbMovers.ResetIterator();
		WHILE THIS^.fbMovers.HasNextObject() DO
			IF ToXpMover(THIS^.fbMovers.GetNextObject(),iTempMover) THEN
				hr := GetMostSignificant(hr, iTempMover.Feedback.HR);
			END_IF
		END_WHILE
		
		IF CheckOk(hr) THEN 
			nSeqDisabling := 50;
		ELSIF FAILED(hr) THEN
			nSeqDisabling := 1000 + nSeqDisabling;
		END_IF			
*)		
		
		
		
	50: // Disable movers
		THIS^.fbMovers.ResetIterator();
		WHILE THIS^.fbMovers.HasNextObject() DO
			IF ToXpMover(THIS^.fbMovers.GetNextObject(),iTempMover) THEN
				hr := GetMostSignificant(hr, iTempMover.Disable());
			END_IF
		END_WHILE
		
		IF CheckOk(hr) THEN 
			nSeqDisabling := 60;
		ELSE
			nSeqDisabling := 1000 + nSeqDisabling;
		END_IF			
		

		
	60: // Disabling movers
		THIS^.fbMovers.ResetIterator();
		WHILE THIS^.fbMovers.HasNextObject() DO
			IF ToXpMover(THIS^.fbMovers.GetNextObject(),iTempMover) THEN
				hr := GetMostSignificant(hr, iTempMover.Feedback.HR);
			END_IF
		END_WHILE
		
		IF CheckOk(hr) THEN 
			nSeqDisabling := 61;
		ELSIF FAILED(hr) THEN
			nSeqDisabling := 1000 + nSeqDisabling;
		END_IF		


	61: // Reset track
		THIS^.fbTracks.ResetIterator();
		WHILE THIS^.fbTracks.HasNextObject() DO
			IF ToXpTrack(THIS^.fbTracks.GetNextObject(),iTempTrack) THEN
				hr := GetMostSignificant(hr, iTempTrack.Reset());
			END_IF
		END_WHILE
		
		IF CheckOk(hr) THEN 
			nSeqDisabling := 62;
		ELSE
			nSeqDisabling := 1000 + nSeqDisabling;
		END_IF		
		
		
	62: // Resetting track
		THIS^.fbTracks.ResetIterator();
		WHILE THIS^.fbTracks.HasNextObject() DO
			IF ToXpTrack(THIS^.fbTracks.GetNextObject(),iTempTrack) THEN
				hr := GetMostSignificant(hr, iTempTrack.Feedback.HR);
			END_IF
		END_WHILE
		
		IF CheckOk(hr) THEN 
			nSeqDisabling := 63;
		ELSIF FAILED(hr) THEN
			nSeqDisabling := 1000 + nSeqDisabling;
		END_IF	

				
	63: // Reset group
		hr := ipGroup.Reset();
		
		IF CheckOk(hr) THEN 
			nSeqDisabling := 64;
		ELSE
			nSeqDisabling := 1000 + nSeqDisabling;
		END_IF		
		
		
	64: // Resetting group
		hr := ipGroup.Feedback.HR;
		
		IF CheckOk(hr) THEN 
			nSeqDisabling := 70;
		ELSIF FAILED(hr) THEN
			nSeqDisabling := 1000 + nSeqDisabling;
		END_IF		
		
		
		

   70: // Disable tracks
		THIS^.fbTracks.ResetIterator();
		WHILE THIS^.fbTracks.HasNextObject() DO
			IF ToXpTrack(THIS^.fbTracks.GetNextObject(),iTempTrack) THEN
				hr := GetMostSignificant(hr, iTempTrack.Disable());
			END_IF
		END_WHILE
		
		IF CheckOk(hr) THEN 
			nSeqDisabling := 80;
		ELSE
			nSeqDisabling := 1000 + nSeqDisabling;
		END_IF			
   
		
   80: // Disabling tracks
		THIS^.fbTracks.ResetIterator();
		WHILE THIS^.fbTracks.HasNextObject() DO
			IF ToXpTrack(THIS^.fbTracks.GetNextObject(),iTempTrack) THEN
				hr := GetMostSignificant(hr, iTempTrack.Feedback.HR);
			END_IF
		END_WHILE
		
		IF CheckOk(hr) THEN 
			nSeqDisabling := 90;
		ELSIF FAILED(hr) THEN
			nSeqDisabling := 1000 + nSeqDisabling;
		END_IF	
				

	90: // Disable group
		hr := ipGroup.Disable();
		
		IF CheckOk(hr) THEN 
			nSeqDisabling := 100;
		ELSE
			nSeqDisabling := 1000 + nSeqDisabling;
		END_IF	
		
		
   100: // Disabling group
		hr := ipGroup.Feedback.HR;
		
		IF CheckOk(hr) THEN 
			nSeqDisabling := 105;
		ELSIF FAILED(hr) THEN
			nSeqDisabling := 1000 + nSeqDisabling;
		END_IF	

		
  105: // Remove tracks from group
		THIS^.fbTracks.ResetIterator();
		WHILE THIS^.fbTracks.HasNextObject() DO
			IF ToXpTrack(THIS^.fbTracks.GetNextObject(),iTempTrack) THEN
				hr := GetMostSignificant(hr, iTempTrack.RemoveFromGroup());
			END_IF
		END_WHILE
		
		IF CheckOk(hr) THEN 
			nSeqDisabling := 106;
		ELSE
			nSeqDisabling := 1000 + nSeqDisabling;
		END_IF			
   
		
   106: // Removing tracks from group
		THIS^.fbTracks.ResetIterator();
		WHILE THIS^.fbTracks.HasNextObject() DO
			IF ToXpTrack(THIS^.fbTracks.GetNextObject(),iTempTrack) THEN
				bOk := bOk AND iTempTrack.PlanarTrack.MCTOPLC_STD.GroupOID = 0;
			END_IF
		END_WHILE
		
		IF bOk THEN 
			nSeqDisabling := 110;
		END_IF	
		
		
	110: // Remove movers from group
		THIS^.fbMovers.ResetIterator();
		WHILE THIS^.fbMovers.HasNextObject() DO
			IF ToXpMover(THIS^.fbMovers.GetNextObject(),iTempMover) THEN
				hr := GetMostSignificant(hr, iTempMover.RemoveFromGroup());
			END_IF
		END_WHILE
		
		IF CheckOk(hr) THEN 
			nSeqDisabling := 120;
		ELSE
			nSeqDisabling := 1000 + nSeqDisabling;
		END_IF		
	
		
	120: // Removing movers from group
		THIS^.fbMovers.ResetIterator();
		WHILE THIS^.fbMovers.HasNextObject() DO
			IF ToXpMover(THIS^.fbMovers.GetNextObject(),iTempMover) THEN
				bOk := bOk AND iTempMover.PlanarMover.MCTOPLC.STD.GroupOID = 0;
			END_IF
		END_WHILE
		
		IF bOk THEN 
			nSeqDisabling := 130;
		END_IF		
	
		
	130: // Remove envirement from group
		hr := ipEnvironment.RemoveFromGroup();
		
		IF CheckOk(hr) THEN 
			nSeqDisabling := 140;
		ELSE
			nSeqDisabling := 1000 + nSeqDisabling;
		END_IF		
		
		
   140: // Removing envirement from group
		hr := ipEnvironment.Feedback.HR;
	
		IF CheckOk(hr) THEN 
			nSeqDisabling := SEQ_DONE;
		ELSIF FAILED(hr) THEN
			nSeqDisabling := 1000 + nSeqDisabling;
		END_IF	
		
	
   SEQ_DONE: //Done
   		Disabling := S_OK;

		
	1000..1999://Error
		hr := GetMostSignificant(hrLastCycle, E_FAIL);

END_CASE

//store last information
hrLastCycle := hr;

// Propagate error
IF FAILED(hr) THEN
	Disabling := hr;
END_IF
END_METHOD

METHOD Enable : CHALET_BaseComponents.I_CH_Feedback
VAR_INPUT
END_VAR
IF NOT THIS^.fbFeedback.Done THEN
	//Error active/not ready
	THIS^.fbFeedback.LastCommandAccepted 	:= FALSE;

ELSIF nSeqEnabling <> 0 THEN
	//System is partial or full enabled. Disable first.
	THIS^.fbFeedback.LastCommandAccepted 	:= FALSE;
ELSE
	THIS^.nSeqDisabling 	:= 0;
	THIS^.nSeqEnabling 		:= 1;
	
	THIS^.eActiveCommand 				:= CHALET_NC.E_NcAxisCommands.Enable;
	THIS^.fbFeedback.LastCommandAccepted:= TRUE;		
	THIS^.fbFeedback.Busy 				:= TRUE;	
END_IF

Enable := THIS^.fbFeedback;
END_METHOD

{attribute 'monitoring':='call'}
PROPERTY Enabled : BOOL
GET
Enabled := nSeqEnabling = SEQ_DONE;
END_GET
END_PROPERTY

METHOD PROTECTED Enabling : HRESULT
VAR
	hr : HRESULT;
	bWatchDogActive : BOOL;
	ipTempMover : I_XP_Mover;
	ipTempMoverPlc : I_XP_Mover_PLC;
	ipTempStation : I_XP_Station;
	ipTempTrack : I_XP_Track;
	
	lrCRotationShortestPos : LREAL;
	bOk : BOOL;
	nSupSeq : UINT;
	nIdx : UINT;
	sMoverType : STRING;
	fDistLastToSet : LREAL;
	fMaxError : LREAL;
	nMoversDetected, nMoverExpected : UDINT;
	bMoverIsMissing : BOOL;
	eMoverDetectionStatus : MoverDetectionStatus;
	stCoordMoverCommStatus : CoordinatedMoverCommStatus;
END_VAR

VAR_INST
	{attribute 'hide'}	
	fbTimeOutSeq : TON; 
	{attribute 'hide'}	
	hrLastCycle 	: HRESULT;
	{attribute 'hide'}	
	nlastState	: UINT;
	
	{attribute 'hide'}	
	fbTimeOutEnabling : FB_TcAlarm;
	{attribute 'hide'}	
	fbErrorEnabling : FB_TcAlarm;
	{attribute 'hide'}	
	fbErrorMoverDetection : FB_TcAlarm;
END_VAR
Enabling := S_PENDING;
CASE nSeqEnabling OF
	0: // Idle
		Enabling := S_OK;	
		
	1: //Redetect all movers on real system
		//timeout is monitored in this sequence
		bWatchDogActive := TRUE;
		
		//check if all mover are present
		THIS^.fbMovers.ResetIterator();
		WHILE THIS^.fbMovers.HasNextObject() DO
			IF ToXpMover(THIS^.fbMovers.GetNextObject(),ipTempMover) AND_THEN ipTempMover.MoverIsNotPresent THEN
				bMoverIsMissing := TRUE;
			END_IF
		END_WHILE
		
		//Decide whether a mover detection should be made or not
		IF (THIS^.ipEnvironment.UtilityEnvirement.XpuTcIo(1).GetOperationMode() = OperationMode.Normal) AND bMoverIsMissing THEN
			THIS^.ipEnvironment.UtilityEnvirement.XpuTcIo(1).SetStartMoverRedetection();
			nSeqEnabling := 5;
		ELSE
			//Skip in simulation
			nSeqEnabling := 30;
		END_IF

	2: //Wait for finish redetection
		//timeout is monitored in this sequence
		bWatchDogActive := TRUE;
		
		eMoverDetectionStatus := THIS^.Enviroment.ProcessingUnitMoverDetectionStatus;
		IF (eMoverDetectionStatus = MoverDetectionStatus.DetectionSuccessful) THEN
			//Done
			nSeqEnabling := 5;
		END_IF

		
	5: //Compare detectet and expectet movers	
	   //timeout is monitored in this sequence
		bWatchDogActive := TRUE;
		
		FOR nIdx := 0 TO 5 DO
			CASE nIdx OF
				0:  sMoverType		:= 'APM4220';
					nMoverExpected 	:= THIS^.ipEnvironment.UtilityEnvirement.XpuTcIo(1).GetMoverDetectionInfos().APM4220Expected;
					nMoversDetected := THIS^.ipEnvironment.UtilityEnvirement.XpuTcIo(1).GetMoverDetectionInfos().APM4220Detected;
				1: 	sMoverType		:= 'APM4221';
					nMoverExpected 	:= THIS^.ipEnvironment.UtilityEnvirement.XpuTcIo(1).GetMoverDetectionInfos().APM4221Expected;
					nMoversDetected := THIS^.ipEnvironment.UtilityEnvirement.XpuTcIo(1).GetMoverDetectionInfos().APM4221Detected;
				2:  sMoverType		:= 'APM4330';
					nMoverExpected 	:= THIS^.ipEnvironment.UtilityEnvirement.XpuTcIo(1).GetMoverDetectionInfos().APM4330Expected;
					nMoversDetected := THIS^.ipEnvironment.UtilityEnvirement.XpuTcIo(1).GetMoverDetectionInfos().APM4330Detected;
				3:  sMoverType		:= 'APM4550';
					nMoverExpected 	:= THIS^.ipEnvironment.UtilityEnvirement.XpuTcIo(1).GetMoverDetectionInfos().APM4550Expected;
					nMoversDetected := THIS^.ipEnvironment.UtilityEnvirement.XpuTcIo(1).GetMoverDetectionInfos().APM4550Detected;
				4:  sMoverType		:= 'total mover count';
					nMoverExpected 	:= THIS^.ipEnvironment.UtilityEnvirement.XpuTcIo(1).GetMoverDetectionInfos().TotalExpected;
					nMoversDetected := THIS^.ipEnvironment.UtilityEnvirement.XpuTcIo(1).GetMoverDetectionInfos().TotalDetected;
					
				5: //Succesfull finished
					nSeqEnabling := 20;	
			END_CASE	

			IF nMoverExpected <> nMoversDetected THEN
				//Error
				nSeqEnabling := 1000 + nSeqEnabling;
				fbErrorMoverDetection.CreateEx(stEventEntry:=TC_EVENTS.CHALET_XPlanar_Events.MoverDetectionFailed, ipSourceInfo := THIS^.fbSourceInfo, bWithConfirmation := FALSE);
				//Mover detection failed. Expected {0} found {1} of type {2}
				fbErrorMoverDetection.ipArguments.AddUDInt(nMoverExpected).AddUDInt(nMoversDetected).AddStringByValue(sMoverType);
				fbErrorMoverDetection.Raise(0);
				EXIT;
			END_IF		
		END_FOR
		
	
	
	10: //Deside if or if not to get orientation of mover. Require an APM9001-0000-4xxx | XPlanar-ID-Bumper
		bWatchDogActive := TRUE;
		IF XPlanarParameterlist.B_GET_MOVER_ORIENTATION AND (THIS^.ipEnvironment.UtilityEnvirement.XpuTcIo(1).GetOperationMode() = OperationMode.Normal) THEN
			nSeqEnabling := 12;
		ELSE
			nSeqEnabling := 20;
		END_IF	
	
	12: //start identification in process
		bWatchDogActive := TRUE;
		 THIS^.ipEnvironment.UtilityEnvirement.XpuTcIo(1).SetCoordMoverCommunicationCmd(CoordinatedMoverCommCommand.IdentifyAndAssignPossible);
		nSeqEnabling:= 13;		
			
	13: // Check for identification in process
		bWatchDogActive := TRUE;
		stCoordMoverCommStatus :=  THIS^.ipEnvironment.UtilityEnvirement.XpuTcIo(1).GetCoordMoverCommStatus();
		IF stCoordMoverCommStatus = CoordinatedMoverCommStatus.CommunicationInProcess THEN
			nSeqEnabling:=14;	
		END_IF
		
	14: // Check result of mover identification
		bWatchDogActive := TRUE;
		stCoordMoverCommStatus :=  THIS^.ipEnvironment.UtilityEnvirement.XpuTcIo(1).GetCoordMoverCommStatus();
		IF stCoordMoverCommStatus = CoordinatedMoverCommStatus.CommunicationSuccessful THEN
			nSeqEnabling := 15;
		ELSIF stCoordMoverCommStatus = CoordinatedMoverCommStatus.CommunicationFailed THEN
		// Error: Identification failed
			nSeqEnabling := 1000 + nSeqEnabling;
		END_IF
		
	15://Determine The orientaion
		bWatchDogActive := TRUE;
		THIS^.ipEnvironment.UtilityEnvirement.XpuTcIo(1).SetCoordMoverCommunicationCmd(CoordinatedMoverCommCommand.DetermineOrientations);
		nSeqEnabling:= 16;
		
	16: // Check for identification in process
		bWatchDogActive := TRUE;
		stCoordMoverCommStatus :=  THIS^.ipEnvironment.UtilityEnvirement.XpuTcIo(1).GetCoordMoverCommStatus();
		IF stCoordMoverCommStatus = CoordinatedMoverCommStatus.CommunicationInProcess THEN
			nSeqEnabling := 17;
		END_IF
		
	17: // Check result of mover identification
		bWatchDogActive := TRUE;
		stCoordMoverCommStatus :=  THIS^.ipEnvironment.UtilityEnvirement.XpuTcIo(1).GetCoordMoverCommStatus();
		IF stCoordMoverCommStatus = CoordinatedMoverCommStatus.CommunicationSuccessful THEN
			nSeqEnabling := 20;
		ELSIF stCoordMoverCommStatus = CoordinatedMoverCommStatus.CommunicationFailed THEN
		// Error: Identification failed
			nSeqEnabling := 1000 + nSeqEnabling;
		END_IF		
		
		
		
		
	20: // Reset movers
		bWatchDogActive := TRUE;
		THIS^.fbMovers.ResetIterator();
		WHILE THIS^.fbMovers.HasNextObject() DO
			IF ToXpMover(THIS^.fbMovers.GetNextObject(),ipTempMover) THEN
				hr := GetMostSignificant(hr, ipTempMover.Reset());
			END_IF
		END_WHILE
		
		IF CheckOk(hr) THEN 
			nSeqEnabling := 21;
		ELSE
			nSeqEnabling := 1000 + nSeqEnabling;
		END_IF		

	21: // Resetting movers
		bWatchDogActive := TRUE;
		THIS^.fbMovers.ResetIterator();
		WHILE THIS^.fbMovers.HasNextObject() DO
			IF ToXpMover(THIS^.fbMovers.GetNextObject(),ipTempMover) THEN
				hr := GetMostSignificant(hr, ipTempMover.Feedback.HR);
			END_IF
		END_WHILE
		
		IF CheckOk(hr) THEN 
			nSeqEnabling := 30;
		ELSIF FAILED(hr) THEN
			nSeqEnabling := 1000 + nSeqEnabling;
		END_IF

		
		
	30: // Configure environment
		bWatchDogActive := TRUE;
		hr := ipEnvironment.Configure();
		
		IF CheckOk(hr) THEN 
			nSeqEnabling := 31;
		ELSE
			nSeqEnabling := 1000 + nSeqEnabling;
		END_IF	

	31: // Configuring environment
		bWatchDogActive := TRUE;
		hr := ipEnvironment.Feedback.HR;
		
		IF CheckOk(hr) THEN 
			nSeqEnabling := 50;
		ELSIF FAILED(hr) THEN
			nSeqEnabling := 1000 + nSeqEnabling;
		END_IF
		
		
	50: //Deside if or if not add enviroment to group
		bWatchDogActive := TRUE;
		IF XPlanarParameterlist.B_ADD_ENVIROMENT_TO_GROUP THEN
			nSeqEnabling := 51;
		ELSE
			nSeqEnabling := 70;
		END_IF
		
	51: // Add environment to group
		bWatchDogActive := TRUE;
		hr := ipEnvironment.AddToGroup(ipGroup);
		
		IF CheckOk(hr) THEN 
			nSeqEnabling := 52;
		ELSE
			nSeqEnabling := 1000 + nSeqEnabling;
		END_IF		

	52: // Adding environment to group
		bWatchDogActive := TRUE;
		hr := ipEnvironment.Feedback.HR;
		
		IF CheckOk(hr) THEN 
			nSeqEnabling := 70;
		ELSIF FAILED(hr) THEN
			nSeqEnabling := 1000 + nSeqEnabling;
		END_IF

		
	70: // Configure the tracks |
		bWatchDogActive := TRUE;
		THIS^.fbTracks.ResetIterator();
		WHILE THIS^.fbTracks.HasNextObject() DO
			IF ToXpTrack(THIS^.fbTracks.GetNextObject(),ipTempTrack) THEN
				hr := GetMostSignificant(hr, ipTempTrack.Configure());
			END_IF
		END_WHILE
		
		IF CheckOk(hr) THEN 
			nSeqEnabling := 71;
		ELSE
			nSeqEnabling := 1000 + nSeqEnabling;
		END_IF	
		
	71: // Configuring the tracks 
		bWatchDogActive := TRUE;
		THIS^.fbTracks.ResetIterator();
		WHILE THIS^.fbTracks.HasNextObject() DO
			IF ToXpTrack(THIS^.fbTracks.GetNextObject(),ipTempTrack) THEN
				hr := GetMostSignificant(hr, ipTempTrack.Configuring());
			END_IF
		END_WHILE
		
		IF CheckOk(hr) THEN 
			nSeqEnabling := 80;
		ELSIF FAILED(hr) THEN
			nSeqEnabling := 1000 + nSeqEnabling;
		END_IF	
		
		
	80: // Enable the tracks
		bWatchDogActive := TRUE;
		THIS^.fbTracks.ResetIterator();
		WHILE THIS^.fbTracks.HasNextObject() DO
			IF ToXpTrack(THIS^.fbTracks.GetNextObject(),ipTempTrack) THEN
				hr := GetMostSignificant(hr, ipTempTrack.Enable());
			END_IF
		END_WHILE
		
		IF CheckOk(hr) THEN 
			nSeqEnabling := 81;
		ELSE
			nSeqEnabling := 1000 + nSeqEnabling;
		END_IF		

	81: // Enabling the tracks
		bWatchDogActive := TRUE;
		THIS^.fbTracks.ResetIterator();
		WHILE THIS^.fbTracks.HasNextObject() DO
			IF ToXpTrack(THIS^.fbTracks.GetNextObject(),ipTempTrack) THEN
				hr := GetMostSignificant(hr, ipTempTrack.Feedback.HR);
			END_IF
		END_WHILE
		
		IF CheckOk(hr) THEN 
			nSeqEnabling := 90;
		ELSIF FAILED(hr) THEN
			nSeqEnabling := 1000 + nSeqEnabling;
		END_IF	
		
	90: //Deside if or if not add tracks to group
		bWatchDogActive := TRUE;
		IF XPlanarParameterlist.B_ADD_TRACKS_TO_GROUP THEN
			nSeqEnabling := 91;
		ELSE
			nSeqEnabling := 95;
		END_IF	
		
	91: // Add tracks to group
		bWatchDogActive := TRUE;
		THIS^.fbTracks.ResetIterator();
		WHILE THIS^.fbTracks.HasNextObject() DO
			IF ToXpTrack(THIS^.fbTracks.GetNextObject(),ipTempTrack) THEN
				hr := GetMostSignificant(hr, ipTempTrack.AddToGroup(ipGroup));
			END_IF
		END_WHILE
		
		IF CheckOk(hr) THEN 
			nSeqEnabling := 92;
		ELSE
			nSeqEnabling := 1000 + nSeqEnabling;
		END_IF	

	92: // Adding tracks to group
		bWatchDogActive := TRUE;
		THIS^.fbTracks.ResetIterator();
		WHILE THIS^.fbTracks.HasNextObject() DO
			IF ToXpTrack(THIS^.fbTracks.GetNextObject(),ipTempTrack) THEN
				hr := GetMostSignificant(hr, ipTempTrack.Feedback.HR);
			END_IF
		END_WHILE
		
		IF CheckOk(hr) THEN 
			nSeqEnabling := 95;
		ELSIF FAILED(hr) THEN
			nSeqEnabling := 1000 + nSeqEnabling;
		END_IF		
	
	95: //Clear list of all paths
		bWatchDogActive := TRUE;
		THIS^.fbPaths.Clear();
		nSeqEnabling := 100;
		

	100..199: // Config Station
	(* All stations are always active to the same step to ensure that all data is available in the next step.
	   The following 100 steps are defined in the station. This makes overwriting easier *)
	   
		bWatchDogActive := TRUE;
		nSupSeq := nSeqEnabling - 100;
		THIS^.fbStations.ResetIterator();
		WHILE THIS^.fbStations.HasNextObject() DO
			IF ToXpStation(THIS^.fbStations.GetNextObject(),ipTempStation) THEN
				//Call this Methode whith seq 0->99, and wait each step until S_OK is returned. Call agaiin on S_Pending
				hr := GetMostSignificant(hr, ipTempStation.Configure(nSupSeq));
			END_IF
		END_WHILE	   
	   
	   
	   	IF CheckOk(hr) AND nSupSeq >= 99 THEN
			//All steps done 
			nSeqEnabling := 205;
		ELSIF FAILED(hr) THEN
			//Error
			nSeqEnabling := 1000 + nSeqEnabling;
		ELSIF CheckOk(hr) THEN 	 
			//active step is done, continous with next
			nSeqEnabling := nSeqEnabling + 1;
		END_IF	


		
	205: //Generate a list of all paths
		bWatchDogActive := TRUE;
		THIS^.fbStations.ResetIterator();
		WHILE THIS^.fbStations.HasNextObject() DO
			IF ToXpStation(THIS^.fbStations.GetNextObject(),ipTempStation) THEN
				THIS^.fbPaths.AddList(ipTempStation.PathsAhead);
			END_IF
		END_WHILE			
		
		nSeqEnabling := 210;
		
	210: // Enable movers
		bWatchDogActive := TRUE;
		THIS^.fbMovers.ResetIterator();
		WHILE THIS^.fbMovers.HasNextObject() DO
			IF ToXpMover(THIS^.fbMovers.GetNextObject(),ipTempMover) THEN
				hr := GetMostSignificant(hr, ipTempMover.Enable());
			END_IF
		END_WHILE
		
		IF CheckOk(hr) THEN 
			nSeqEnabling := 211;
		ELSE
			nSeqEnabling := 1000 + nSeqEnabling;
		END_IF	
		
	211: // Enabling movers
		bWatchDogActive := TRUE;
		THIS^.fbMovers.ResetIterator();
		WHILE THIS^.fbMovers.HasNextObject() DO
			IF ToXpMover(THIS^.fbMovers.GetNextObject(),ipTempMover) THEN
				hr := GetMostSignificant(hr, ipTempMover.Feedback.HR);
			END_IF
		END_WHILE
		
		IF CheckOk(hr) THEN 
			nSeqEnabling := 220;
		ELSIF FAILED(hr) THEN
			nSeqEnabling := 1000 + nSeqEnabling;
		END_IF	
		

	220: //Rotate A-Axis to zero
		bWatchDogActive := TRUE;
		THIS^.fbMovers.ResetIterator();
		WHILE THIS^.fbMovers.HasNextObject() DO
			IF ToXpMover(THIS^.fbMovers.GetNextObject(),ipTempMover) THEN
				hr := GetMostSignificant(hr, ipTempMover.MoveA(0));
			END_IF
		END_WHILE
		
		IF CheckOk(hr) THEN 
			nSeqEnabling := 221;
		ELSE
			nSeqEnabling := 1000 + nSeqEnabling;
		END_IF	
		
	221: //Rotating A-Axis to Zero	
		bWatchDogActive := TRUE;		
		THIS^.fbMovers.ResetIterator();
		WHILE THIS^.fbMovers.HasNextObject() DO
			IF ToXpMover(THIS^.fbMovers.GetNextObject(),ipTempMover) THEN
				hr := GetMostSignificant(hr, ipTempMover.Feedback.HR);
			END_IF
		END_WHILE
		
		IF CheckOk(hr) THEN 
			nSeqEnabling := 222;
		ELSIF FAILED(hr) THEN
			nSeqEnabling := 1000 + nSeqEnabling;
		END_IF	
		
		
		
	222: //Rotate B-Axis to zero
		bWatchDogActive := TRUE;
		THIS^.fbMovers.ResetIterator();
		WHILE THIS^.fbMovers.HasNextObject() DO
			IF ToXpMover(THIS^.fbMovers.GetNextObject(),ipTempMover) THEN
				hr := GetMostSignificant(hr, ipTempMover.MoveB(0));
			END_IF
		END_WHILE
		
		IF CheckOk(hr) THEN 
			nSeqEnabling := 223;
		ELSE
			nSeqEnabling := 1000 + nSeqEnabling;
		END_IF	
		
	223: //Rotating B-Axis to zero
		bWatchDogActive := TRUE;			
		THIS^.fbMovers.ResetIterator();
		WHILE THIS^.fbMovers.HasNextObject() DO
			IF ToXpMover(THIS^.fbMovers.GetNextObject(),ipTempMover) THEN
				hr := GetMostSignificant(hr, ipTempMover.Feedback.HR);
			END_IF
		END_WHILE
		
		IF CheckOk(hr) THEN 
			nSeqEnabling := 230;
		ELSIF FAILED(hr) THEN
			nSeqEnabling := 1000 + nSeqEnabling;
		END_IF		
		
				
		
	230: //Rotate C-Axis to "Zero" (to the next 90 degree pitch)
		bWatchDogActive := TRUE;
		THIS^.fbMovers.ResetIterator();
		WHILE THIS^.fbMovers.HasNextObject() DO
			IF ToXpMover(THIS^.fbMovers.GetNextObject(),ipTempMover) THEN
				// Decide which 90 degree pitch is closer to the current position. If the remainder is greater than 45 degrees, then round up to the next 90 degree division.
				lrCRotationShortestPos := DINT_TO_LREAL(LREAL_TO_DINT(ipTempMover.PlanarMover.MCTOPLC.SET.SetPos.C / 90.0) * 90);
				lrCRotationShortestPos := MODABS(	lr_Value := lrCRotationShortestPos, 
													lr_Arg := ipTempMover.CAxisModulo);
				hr := GetMostSignificant(hr, ipTempMover.MoveC(	fPosition		:= lrCRotationShortestPos, 
																additionalTurns := 0,
																direction		:= Tc3_Mc3Definitions.MC_DIRECTION.mcDirectionShortestWay));
			END_IF
		END_WHILE
		
		IF CheckOk(hr) THEN 
			nSeqEnabling := 231;
		ELSE
			nSeqEnabling := 1000 + nSeqEnabling;
		END_IF	
		
		
	231: //Rotating C-Axis to Zero		
		bWatchDogActive := TRUE;	
		THIS^.fbMovers.ResetIterator();
		WHILE THIS^.fbMovers.HasNextObject() DO
			IF ToXpMover(THIS^.fbMovers.GetNextObject(),ipTempMover) THEN
				hr := GetMostSignificant(hr, ipTempMover.Feedback.HR);
			END_IF
		END_WHILE
		
		IF CheckOk(hr) THEN 
			nSeqEnabling := 240;
		ELSIF FAILED(hr) THEN
			nSeqEnabling := 1000 + nSeqEnabling;
		END_IF	
		
			
	240: //Deside if or if not add movers to group
		bWatchDogActive := TRUE;
		IF XPlanarParameterlist.B_ADD_MOVERS_TO_GROUP THEN
			nSeqEnabling := 210;
		ELSE
			nSeqEnabling := 300;
		END_IF	
		
	241: // Add movers to group
		bWatchDogActive := TRUE;
		THIS^.fbMovers.ResetIterator();
		WHILE THIS^.fbMovers.HasNextObject() DO
			IF ToXpMover(THIS^.fbMovers.GetNextObject(),ipTempMover) THEN
				hr := GetMostSignificant(hr, ipTempMover.AddToGroup(THIS^.ipGroup));
			END_IF
		END_WHILE
		
		IF CheckOk(hr) THEN 
			nSeqEnabling := 242;
		ELSE
			nSeqEnabling := 1000 + nSeqEnabling;
		END_IF	
		
		
	242: // Adding mover to group
		bWatchDogActive := TRUE;
		THIS^.fbMovers.ResetIterator();
		WHILE THIS^.fbMovers.HasNextObject() DO
			IF ToXpMover(THIS^.fbMovers.GetNextObject(),ipTempMover) THEN
				hr := GetMostSignificant(hr, ipTempMover.Feedback.HR);
			END_IF
		END_WHILE
		
		IF CheckOk(hr) THEN 
			nSeqEnabling := 300;
		ELSIF FAILED(hr) THEN
			nSeqEnabling := 1000 + nSeqEnabling;
		END_IF		
	
		
		
	300: // Enable group
		bWatchDogActive := TRUE;
		hr := ipGroup.Enable();
		
		IF CheckOk(hr) THEN 
			nSeqEnabling := 310;
		ELSE
			nSeqEnabling := 1000 + nSeqEnabling;
		END_IF	
		
	310: // Enabling group
		bWatchDogActive := TRUE;
		hr := ipGroup.Feedback.HR;
		
		IF CheckOk(hr) THEN 
			//nSeqEnabling := 350;
			nSeqEnabling := 400;
		ELSIF FAILED(hr) THEN
			nSeqEnabling := 1000 + nSeqEnabling;
		END_IF	
		
		
//	340: // Check dist last known position to current pos
//		bWatchDogActive := TRUE;
//		THIS^.fbMovers.ResetIterator();
//		WHILE THIS^.fbMovers.HasNextObject() DO
//			IF ToXpMover(THIS^.fbMovers.GetNextObject(),ipTempMover) THEN
//				IF ipTempMover.PositionAtDisable.x <> 0 AND ipTempMover.PositionAtDisable.y <> 0 THEN
//					fDistLastToSet := F_DistXYVectors(ipTempMover.PositionAtDisable, ipTempMover.PositionSet);
//					fMaxError := MAX(fMaxError, fDistLastToSet);
//				END_IF
//			END_IF
//		END_WHILE
//		IF fMaxError < 50 THEN
//			nSeqEnabling := 350;
//		ELSE
//			nSeqEnabling := 400;			
//		END_IF
//
//		
//	350: // Move to last valide known position
//		bWatchDogActive := TRUE;
//		THIS^.fbMovers.ResetIterator();
//		WHILE THIS^.fbMovers.HasNextObject() DO
//			IF ToXpMover(THIS^.fbMovers.GetNextObject(),ipTempMover) THEN
//				IF ipTempMover.PositionAtDisable.x <> 0 AND ipTempMover.PositionAtDisable.y <> 0 THEN
//					hr := GetMostSignificant(hr, ipTempMover.MoveXY(fPosition_X := ipTempMover.PositionAtDisable.x, 
//																	fPosition_Y := ipTempMover.PositionAtDisable.y));
//				END_IF
//			END_IF
//		END_WHILE
//		//Its posible that the command failed. Do not exit SEQ
//		nSeqEnabling := 351;
//
//
//		
//	351: // Wait for standstill
//		bWatchDogActive := TRUE;
//		
//		bOk := TRUE;
//		THIS^.fbMovers.ResetIterator();
//		WHILE THIS^.fbMovers.HasNextObject() DO
//			IF ToXpMover(THIS^.fbMovers.GetNextObject(),ipTempMover) THEN
//				bOk := bOk AND ipTempMover.Standstill;
//			END_IF
//		END_WHILE
//		THIS^.fbMovers.RestoreIterator();
//		
//		IF bOk THEN 
//			nSeqEnabling := 400;
//		END_IF	

		
	400: (*	Restart of the sequenze "JoiningTrack". Default strategy is that each mover joins the closest track
			Outsourced to a method for easier overwriting *)
		THIS^.nSeqJoiningTrack := 0;	
		nSeqEnabling := 401;
	

	401: (*	Default strategy is that each mover joins the closest track
			Outsourced to a method for easier overwriting *)
		hr := THIS^.JoiningTrack();

		IF CheckOk(hr) THEN 
			nSeqEnabling := 500;
		ELSIF FAILED(hr) THEN
			nSeqEnabling := 1000 + nSeqEnabling;
		END_IF	
		
	

	
	500: (*	Restart of the sequenze "JoiningStation" to distribute the movers to the available stations.
			Outsourced to a method for easier overwriting *)
		THIS^.nSeqJoiningStation := 0;	
		nSeqEnabling := 501;	
	
	501: (*	Distribute the movers to the available stations.
		 	Outsourced to a method for easier overwriting *)
		hr := THIS^.JoiningStation();

		IF CheckOk(hr) THEN 
			nSeqEnabling := SEQ_DONE;
		ELSIF FAILED(hr) THEN
			nSeqEnabling := 1000 + nSeqEnabling;
		END_IF	

		
	SEQ_DONE: // Done
		Enabling := S_OK;

		
	1000..1999://Error
		hr := GetMostSignificant(hrLastCycle, E_FAIL);
		//Only rais if timeout is not active
		IF NOT fbErrorEnabling.bRaised AND NOT fbTimeOutEnabling.bRaised THEN 
			fbErrorEnabling.CreateEx(stEventEntry:=TC_EVENTS.CHALET_Base_Events.ErrorEnabling, ipSourceInfo := THIS^.fbSourceInfo, bWithConfirmation := FALSE);
			fbErrorEnabling.ipArguments.AddUInt(nSeqEnabling-1000);
			fbErrorEnabling.Raise(0);
		END_IF
END_CASE


//Timeout after to long stay in one of the following seq.
fbTimeOutSeq.IN := (nlastState = nSeqEnabling) AND bWatchDogActive;
fbTimeOutSeq.PT := T#10S;
fbTimeOutSeq();
nlastState := nSeqEnabling;

IF fbTimeOutSeq.Q THEN
	IF NOT fbTimeOutEnabling.bRaised THEN 
		fbTimeOutEnabling.CreateEx(stEventEntry:=TC_EVENTS.CHALET_Base_Events.TimeOutEnabling, ipSourceInfo := THIS^.fbSourceInfo, bWithConfirmation := FALSE);
		fbTimeOutEnabling.ipArguments.AddUInt(nSeqEnabling);
		fbTimeOutEnabling.Raise(0);
	END_IF
	//next seq is error
	nSeqEnabling := 1000 + nSeqEnabling;
END_IF

//Clear Tc3-Eventlogger alarm 
IF nSeqEnabling <= SEQ_DONE THEN
	fbTimeOutEnabling.Clear(0,0);
	fbErrorEnabling.Clear(0,0);
	fbErrorMoverDetection.Clear(0,0);
END_IF


//store last information
hrLastCycle := hr;

// Propagate error
IF FAILED(hr) THEN
	Enabling := hr;
END_IF
END_METHOD

METHOD FastStop : I_CH_Feedback
VAR
	ipMoverPlc : I_XP_Mover_PLC;
END_VAR
THIS^.Movers.ResetIterator();
WHILE THIS^.Movers.HasNextObject() DO
	IF __QUERYINTERFACE(THIS^.Movers.GetNextObject(),ipMoverPlc) THEN
		//Change deceleration to MC_MAXIMUM for each mover
		ipMoverPlc.SetDynConstraint_Path(V:= MC_DEFAULT, A:= MC_DEFAULT, D:= MC_MAXIMUM, J:= MC_MAXIMUM);
	END_IF
END_WHILE
THIS^.Movers.RestoreIterator();


FastStop := THIS^.Disable();
THIS^.Disabling();
END_METHOD

METHOD Initialize : HRESULT
VAR_INPUT
END_VAR
VAR
	hr 				: HRESULT := S_OK;
	ipEachStation 	: I_XP_Station;
END_VAR
VAR_INST
	//This error cannot be reset. Requires a reset cold
	{attribute 'hide'}	
	fbInitError : FB_TcAlarm;
	{attribute 'hide'}	
	fbMissingInterfaceAlarm : FB_TcAlarm;
END_VAR
//Set to busy on first call
IF THIS^.eActiveCommand <> CHALET_NC.E_NcAxisCommands.Initialize THEN
	THIS^.eActiveCommand 					:= CHALET_NC.E_NcAxisCommands.Initialize;
	THIS^.fbFeedback.LastCommandAccepted	:= TRUE;		
	THIS^.fbFeedback.Busy 					:= TRUE;
END_IF




//Check Error during FB_Init
IF THIS^.bErrorDuringFbInit THEN
	IF NOT fbInitError.bRaised THEN 
		//This error cannot be reset. Requires a reset cold
		fbInitError.CreateEx(stEventEntry:=TC_EVENTS.CHALET_Base_Events.ErrorFBinit, ipSourceInfo := THIS^.fbSourceInfo, bWithConfirmation := FALSE);
		fbInitError.Raise(0);
	END_IF
	Initialize:= E_FAIL;
	THIS^.fbFeedback.HR := Initialize;
	RETURN;
END_IF	


//Check if Envirement and Group is existing
IF  THIS^.ipGroup = 0 THEN
	IF NOT fbMissingInterfaceAlarm.bRaised THEN 
		//This error cannot be reset. Requires a reset cold
		fbMissingInterfaceAlarm.CreateEx(stEventEntry:=TC_EVENTS.CHALET_XPlanar_Events.MissingGroupe, ipSourceInfo := THIS^.fbSourceInfo, bWithConfirmation := FALSE);
		fbMissingInterfaceAlarm.Raise(0);
	END_IF
	Initialize := E_FAIL;
	THIS^.fbFeedback.HR := Initialize;
	RETURN;
END_IF

//Check if Envirement and Group is existing
IF THIS^.ipEnvironment = 0 THEN
	IF NOT fbMissingInterfaceAlarm.bRaised THEN 
		//This error cannot be reset. Requires a reset cold
		fbMissingInterfaceAlarm.CreateEx(stEventEntry:=TC_EVENTS.CHALET_XPlanar_Events.MissingEnvironment, ipSourceInfo := THIS^.fbSourceInfo, bWithConfirmation := FALSE);
		fbMissingInterfaceAlarm.Raise(0);
	END_IF
	Initialize := E_FAIL;
	THIS^.fbFeedback.HR := Initialize;
	RETURN;
END_IF


//Init envirement first to get access to XPlanar_Utility
IF THIS^.ipEnvironment.Initialize() = S_OK THEN
	hr := GetMostSignificant(hr, THIS^.ipGroup.Initialize());
	hr := GetMostSignificant(hr, THIS^.fbMovers.Initialize());
	hr := GetMostSignificant(hr, THIS^.fbTracks.Initialize());
	hr := GetMostSignificant(hr, THIS^.fbStations.Initialize());
	hr := GetMostSignificant(hr, THIS^.fbTriggers.Initialize());
	hr := GetMostSignificant(hr, THIS^.fbZones.Initialize());
ELSE
	hr := S_PENDING;
END_IF	



THIS^.bInitDone := (hr = S_OK);

Initialize:= hr;

THIS^.fbFeedback.HR := Initialize;
END_METHOD

{attribute 'monitoring':='call'}
PROPERTY Initialized : BOOL
GET
Initialized := bInitDone;
END_GET
END_PROPERTY

METHOD CheckTargetExists : BOOL //Return TRUE if target is existing
VAR_INPUT
	sStation	: STRING; //Group of the targed station or LUID
END_VAR
VAR
	ipEachStation : I_XP_Station_PLC;
END_VAR
THIS^.fbStations.ResetIterator();
WHILE THIS^.fbStations.HasNextObject() DO
	IF __QUERYINTERFACE(THIS^.fbStations.GetNextObject(),ipEachStation) THEN
		//Return TRUE if found
		IF (ipEachStation.TargetGroupe = sStation) OR (ipEachStation.LUID = sStation) THEN
			CheckTargetExists := TRUE;
			EXIT;
		END_IF
	END_IF
END_WHILE
THIS^.fbStations.RestoreIterator();
END_METHOD

//Returns the station that is closest to the point according to Phytagoras
METHOD GetStationClosestTo : I_XP_Station
VAR_INPUT
	pos : MoverVector;
END_VAR
VAR
	stPositionStation : MoverVector;
	ipEachStation : I_XP_Station;
	fTempDist : LREAL;
	fDistClosestStation: LREAL := CHALET_BaseComponents.GVL_Datatypes.cMaxLreal;
END_VAR
THIS^.fbStations.ResetIterator();
WHILE THIS^.fbStations.HasNextObject() DO
	IF __QUERYINTERFACE(THIS^.fbStations.GetNextObject(),ipEachStation) THEN
		stPositionStation.x := ipEachStation.PositionOnTrackXY.x;
		stPositionStation.y := ipEachStation.PositionOnTrackXY.y;
		
		fTempDist := F_DistXYVectors(pos, stPositionStation);
		
		IF fTempDist <= fDistClosestStation THEN
			fDistClosestStation := fTempDist;
			GetStationClosestTo := ipEachStation;
		END_IF
		
	END_IF
END_WHILE
THIS^.fbStations.RestoreIterator();
END_METHOD

METHOD Station : I_XP_Station_PLC
VAR_INPUT
	sLUID : STRING;
END_VAR
//IF no station was found, INTERFACE is 0 -> can generate fatal error
__QUERYINTERFACE(THIS^.fbStations.FindLUID(sLUID),Station);
END_METHOD

METHOD LinkEnvironment : HRESULT
VAR_INPUT
	ipEnvironment : I_CH_Object;
END_VAR

VAR
	ipXpEnvironment : I_XP_Environment;
END_VAR
IF ipEnvironment <> 0 AND_THEN __QUERYINTERFACE(ipEnvironment,ipXpEnvironment) THEN
	THIS^.ipEnvironment := ipXpEnvironment;
ELSE
	LinkEnvironment := E_FAIL;
	THIS^.bErrorDuringFbInit := TRUE;
END_IF
END_METHOD

METHOD LinkGroup : HRESULT
VAR_INPUT
	ipGroup : I_CH_Object;
END_VAR

VAR
	ipXpGroup : I_XP_Group;
END_VAR
IF ipGroup <> 0 AND_THEN __QUERYINTERFACE(ipGroup,ipXpGroup) THEN
	THIS^.ipGroup := ipXpGroup;
ELSE
	LinkGroup := E_FAIL;
	THIS^.bErrorDuringFbInit := TRUE;
END_IF
END_METHOD

METHOD RegisterMover : HRESULT
VAR_INPUT
	ipMover : I_CH_Object;
END_VAR

VAR
	ipXpMover : I_XP_Mover;
END_VAR
IF ipMover = 0 THEN
	//Invalide interface	
	THIS^.bErrorDuringFbInit := TRUE;
	RegisterMover := E_FAIL;
	
ELSIF NOT __QUERYINTERFACE(ipMover, ipXpMover) THEN
	//The required interface is missing
	THIS^.bErrorDuringFbInit := TRUE;
	RegisterMover := E_FAIL;
	
ELSIF THIS^.fbMovers.IsFull THEN
	//List is full
	THIS^.bErrorDuringFbInit := TRUE;
	RegisterMover := E_FAIL;
	
ELSIF THIS^.bInitDone THEN
	//To late. System is initilized
	THIS^.bErrorDuringFbInit := TRUE;
	RegisterMover := E_FAIL;
	
ELSE
	
	THIS^.fbMovers.AddObject(ipMover);
END_IF
END_METHOD

METHOD RegisterStation : HRESULT
VAR_INPUT
	ipStation : I_CH_Object;
END_VAR

VAR
	ipXpStation : I_XP_Station;
END_VAR
IF ipStation = 0 THEN
	//Invalide interface	
	THIS^.bErrorDuringFbInit := TRUE;
	RegisterStation := E_FAIL;
	
ELSIF NOT __QUERYINTERFACE(ipStation, ipXpStation) THEN
	//The required interface is missing
	THIS^.bErrorDuringFbInit := TRUE;
	RegisterStation := E_FAIL;
	
ELSIF THIS^.fbStations.IsFull THEN
	//List is full
	THIS^.bErrorDuringFbInit := TRUE;
	RegisterStation := E_FAIL;
	
ELSIF THIS^.bInitDone THEN
	//To late. System is initilized
	THIS^.bErrorDuringFbInit := TRUE;
	RegisterStation := E_FAIL;
		
ELSE
	
	THIS^.fbStations.AddObject(ipStation);
END_IF
END_METHOD

METHOD RegisterTrack : HRESULT
VAR_INPUT
	ipTrack : I_CH_Object;
END_VAR

VAR
	ipXpTrack : I_XP_Track;
END_VAR
IF ipTrack = 0 THEN
	//Invalide interface	
	THIS^.bErrorDuringFbInit := TRUE;
	RegisterTrack := E_FAIL;
	
ELSIF NOT __QUERYINTERFACE(ipTrack, ipXpTrack) THEN
	//The required interface is missing
	THIS^.bErrorDuringFbInit := TRUE;
	RegisterTrack := E_FAIL;
	
ELSIF THIS^.fbTracks.IsFull THEN
	//List is full
	THIS^.bErrorDuringFbInit := TRUE;
	RegisterTrack := E_FAIL;
	
ELSIF THIS^.bInitDone THEN
	//To late. System is initilized
	THIS^.bErrorDuringFbInit := TRUE;
	RegisterTrack := E_FAIL;
		
ELSE
	
	THIS^.fbTracks.AddObject(ipTrack);
END_IF
END_METHOD

METHOD RegisterTrigger : HRESULT
VAR_INPUT
	ipTrigger	: CHALET_BaseComponents.I_CH_Object;
END_VAR
VAR
	ipXpTrigger : I_Xp_Trigger;
END_VAR
IF ipTrigger = 0 THEN
	//Invalide interface	
	THIS^.bErrorDuringFbInit := TRUE;
	RegisterTrigger := E_FAIL;
	
ELSIF NOT __QUERYINTERFACE(ipTrigger, ipXpTrigger) THEN
	//The required interface is missing
	THIS^.bErrorDuringFbInit := TRUE;
	RegisterTrigger := E_FAIL;
	
ELSIF THIS^.fbTriggers.IsFull THEN
	//List is full
	THIS^.bErrorDuringFbInit := TRUE;
	RegisterTrigger := E_FAIL;
	
ELSIF THIS^.bInitDone THEN
	//To late. System is initilized
	THIS^.bErrorDuringFbInit := TRUE;
	RegisterTrigger := E_FAIL;
		
ELSE
	
	THIS^.fbTriggers.AddObject(ipTrigger);
END_IF
END_METHOD

METHOD RegisterZone : HRESULT
VAR_INPUT
	ipZone	: CHALET_BaseComponents.I_CH_Object;
END_VAR
VAR
	ipXpsZone : I_XP_Zone;
END_VAR
IF ipZone = 0 THEN
	//Invalide interface	
	THIS^.bErrorDuringFbInit := TRUE;
	RegisterZone := E_FAIL;

ELSIF NOT __QUERYINTERFACE(ipZone, ipXpsZone) THEN
	//The required interface is missing
	THIS^.bErrorDuringFbInit := TRUE;
	RegisterZone := E_FAIL;
	
ELSIF THIS^.fbZones.IsFull THEN
	//List is full
	THIS^.bErrorDuringFbInit := TRUE;
	RegisterZone := E_FAIL;
	
ELSIF THIS^.bInitDone THEN
	//To late. System is initilized
	THIS^.bErrorDuringFbInit := TRUE;
	RegisterZone := E_FAIL;
		
ELSE
	
	THIS^.fbZones.AddObject(ipZone);	
END_IF
END_METHOD

METHOD CheckForErrors : BOOL
VAR
	ipEachMover : I_XP_Mover;
	bErrorFound : BOOL;
	bAtLeastOnMoverIsEnabled : BOOL;
END_VAR
VAR_INST
	{attribute 'hide'}
	bErrorFoundOld : BOOL;
END_VAR
THIS^.fbMovers.ResetIterator();
WHILE THIS^.fbMovers.HasNextObject() DO
	IF __QUERYINTERFACE(THIS^.fbMovers.GetNextObject(),ipEachMover) THEN
			bErrorFound := bErrorFound OR ipEachMover.Feedback.Error;
			bErrorFound := bErrorFound OR (ipEachMover.PlanarMover.MCTOPLC.STD.ErrorCode <> 0);
									
			//Only Disable System on Error, if at least on Mover is Enabled
			bAtLeastOnMoverIsEnabled := ipEachMover.Enabled OR bAtLeastOnMoverIsEnabled;
	END_IF
END_WHILE
THIS^.fbMovers.RestoreIterator();

//check this system (Enabling disabling)
bErrorFound := bErrorFound OR THIS^.fbFeedback.Error;


//Do an disable at new error found
IF bAtLeastOnMoverIsEnabled AND bErrorFound AND NOT bErrorFoundOld THEN 
	THIS^.Disable();
END_IF

//Keep information
bErrorFoundOld := bErrorFound;
END_METHOD

{attribute 'monitoring':='call'}
PROPERTY Enviroment : I_XP_Environment
GET
Enviroment := THIS^.ipEnvironment;
END_GET
END_PROPERTY

METHOD FB_init : BOOL
VAR_INPUT
	bInitRetains : BOOL; // if TRUE, the retain variables are initialized (warm start / cold start)
	bInCopyCode : BOOL;  // if TRUE, the instance afterwards gets moved into the copy code (online change)
	
END_VAR
VAR
	fbGetCurTaskIdx  : GETCURTASKINDEX;
END_VAR
END_METHOD

{attribute 'monitoring':='call'}
PROPERTY Feedback : CHALET_BaseComponents.I_CH_Feedback
GET
Feedback := THIS^.fbFeedback;
END_GET
END_PROPERTY

{attribute 'monitoring':='call'}
PROPERTY Movers : CHALET_BaseComponents.I_CH_LIST
GET
Movers := THIS^.fbMovers;
END_GET
END_PROPERTY

{attribute 'monitoring':='call'}
PROPERTY Paths : CHALET_BaseComponents.I_CH_LIST
GET
Paths := THIS^.fbPaths;
END_GET
END_PROPERTY

{attribute 'monitoring':='call'}
PROPERTY Stations : CHALET_BaseComponents.I_CH_LIST
GET
Stations := THIS^.fbStations;
END_GET
END_PROPERTY

//Suppress to change the dynamic(Gap) of passing movers in all stations. This is usefull in startup
PROPERTY SuppressAllDynamicsChanges : BOOL
SET
VAR
	ipTempStationPlc : I_XP_Station_PLC;
END_VAR
// go through the list and write request to it
THIS^.fbStations.ResetIterator();
WHILE THIS^.fbStations.HasNextObject() DO
	IF __QUERYINTERFACE(THIS^.fbStations.GetNextObject(), ipTempStationPlc) THEN
		ipTempStationPlc.SuppressDynamicsChange := SuppressAllDynamicsChanges;
	END_IF
END_WHILE
THIS^.fbStations.RestoreIterator();
END_SET
END_PROPERTY

{attribute 'monitoring':='call'}
PROPERTY Tracks : CHALET_BaseComponents.I_CH_LIST
GET
Tracks := THIS^.fbTracks;
END_GET
END_PROPERTY

{attribute 'monitoring':='call'}
PROPERTY Triggers : CHALET_BaseComponents.I_CH_LIST
GET
Triggers := THIS^.fbTriggers;
END_GET
END_PROPERTY

METHOD Update : HRESULT
VAR
	hr : HRESULT;
END_VAR
//Force to do an init at beginn
IF NOT THIS^.Initialized THEN
	THIS^.Initialize();
	RETURN;
END_IF

hr := S_OK;

hr := GetMostSignificant(hr, THIS^.Enabling());
hr := GetMostSignificant(hr, THIS^.Disabling());




// ********************** Set feedback depending on active command *******************************
IF THIS^.eActiveCommand <> E_NcAxisCommands.None THEN
	fbFeedback.ActiveCommand 	:= TO_STRING(THIS^.eActiveCommand);	
END_IF

CASE THIS^.eActiveCommand OF
	E_NcAxisCommands.None: 
		;

	E_NcAxisCommands.Initialize:
		fbFeedback.Busy 		:= NOT THIS^.bInitDone;
		fbFeedback.Done 		:= THIS^.bInitDone;
		fbFeedback.ErrorId 		:= 0;
		
	E_NcAxisCommands.Enable:
		fbFeedback.Busy 		:= nSeqEnabling > 0;
		fbFeedback.Done 		:= THIS^.Enabled;
		IF nSeqEnabling > 1000 THEN
			fbFeedback.ErrorId 		:= nSeqEnabling;
		END_IF
		
	E_NcAxisCommands.Disable:
		fbFeedback.Busy 		:= nSeqDisabling > 0;
		fbFeedback.Done 		:= THIS^.Disabled;
		IF nSeqDisabling > 1000 THEN
			fbFeedback.ErrorId 		:= nSeqDisabling;
		END_IF
		


	ELSE//External command in subclass
		;
END_CASE


// **********************  Stop to execute commands on .done or .error ***************************
IF fbFeedback.Done OR THIS^.fbFeedback.Error THEN
	eActiveCommand 				:= E_NcAxisCommands.None;
END_IF

CheckForErrors();

hr := GetMostSignificant(hr, THIS^.fbMovers.Update());
hr := GetMostSignificant(hr, THIS^.fbTracks.Update());
hr := GetMostSignificant(hr, THIS^.fbStations.Update());
hr := GetMostSignificant(hr, THIS^.fbZones.Update());
hr := GetMostSignificant(hr, THIS^.fbTriggers.Update());
hr := GetMostSignificant(hr, THIS^.ipGroup.Update());
hr := GetMostSignificant(hr, THIS^.ipEnvironment.Update());


Update:= hr;
END_METHOD

{attribute 'monitoring':='call'}
PROPERTY Zones : CHALET_BaseComponents.I_CH_LIST
GET
Zones := THIS^.fbZones;
END_GET
END_PROPERTY

END_FUNCTION_BLOCK

// FUNCTIONs/F_DistXYVectors
FUNCTION F_DistXYVectors : LREAL
VAR_INPUT
	pos1 : REFERENCE TO MoverVector;
	pos2 : REFERENCE TO MoverVector;
END_VAR
VAR
	fbPos2D : PositionXY;
END_VAR

IF NOT __ISVALIDREF(pos1) OR NOT __ISVALIDREF(pos2) THEN
	//Error
	F_DistXYVectors := -1;
	RETURN;
END_IF

fbPos2D.x := pos1.x - pos2.x;
fbPos2D.y := pos1.y - pos2.y;

F_DistXYVectors := fbPos2D.GetRadius();

END_FUNCTION

// COMPONENTs/Track/FB_XP_Track
{attribute 'no_explicit_call' := 'Do not call the body - Stick to OOP'}
(* XPlanar track - n per associated XPlanar. Can be instantiated as an array and/or individually
	The Planar track is a software object that represents a (virtual) one-dimensional path on the two-dimensional XPlanar stator surface. 
	Several Planar movers can be lined up and moved on this path. Collisions are prevented by keeping a preset distance between the movers. *)	
FUNCTION_BLOCK FB_XP_Track EXTENDS FB_CH_Object IMPLEMENTS I_XP_Track
VAR
	//Link to Planar-Track object
	fbTrack : MC_PlanarTrack;
	
	{attribute 'hide'}  
	bInitDone :BOOL := FALSE;
	{attribute 'hide'}               	
	fbFeedback 			: FB_XP_Feedback(ipSourceInfo := fbSourceInfo);	
	{attribute 'hide'}                   	
	eActiveCommand 		: CHALET_Nc.E_NcAxisCommands := CHALET_Nc.E_NcAxisCommands.None;
	{attribute 'hide'}
	ipXpSystem : I_XP_System_Registration;
	{attribute 'hide'}	
	nSeqConfiguring : UINT;
	{attribute 'hide'} 
	ipTracksEndAtThis : ARRAY[0..(XPlanarParameterlist.N_MAX_STATIONS_AHEAD_OR_BEHIND-1)] OF I_XP_Track;
	{attribute 'hide'} 
	ipTracksStartFromThis : ARRAY[0..(XPlanarParameterlist.N_MAX_STATIONS_AHEAD_OR_BEHIND-1)] OF I_XP_Track;
	{attribute 'hide'}  
	fbListOfStationsOnTrack : FB_CH_List;

	{attribute 'hide'}  
	bIsClosedLoop : BOOL;
	{attribute 'hide'}  
	PreviousTrackOTCIDs 	: ARRAY[0..(XPlanarParameterlist.N_MAX_STATIONS_AHEAD_OR_BEHIND-1)] OF OTCID;
	{attribute 'hide'}  
	SubsequentTrackOTCIDs 	: ARRAY[0..(XPlanarParameterlist.N_MAX_STATIONS_AHEAD_OR_BEHIND-1)] OF OTCID;
	
	{attribute 'hide'}
	fbListOfMoversOnTrack : FB_CH_List;
	{attribute 'hide'}  
	fbTracksAhead : FB_CH_List;
	{attribute 'hide'}  
	fbTracksBehinde : FB_CH_List;
	

	{attribute 'hide'}  
	fbListPathsOnThisTrack : FB_CH_List;	
	
END_VAR

// Planar-Feedback objects
VAR
	{attribute 'hide'} 
	fbFeedbackDisable: MC_PlanarFeedback;
	{attribute 'hide'} 
	fbFeedbackEnable : MC_PlanarFeedback;
	{attribute 'hide'} 
	fbFeedbackAddToGrp : MC_PlanarFeedback;
	{attribute 'hide'} 
	fbFeedbackRmvFromGrp : MC_PlanarFeedback;
	{attribute 'hide'} 
	fbFeedbackReset : MC_PlanarFeedback;
END_VAR

METHOD Configure : HRESULT // This is called once during system enabling
VAR_INPUT
END_VAR
VAR_INST
	{attribute 'hide'}  
	fbAlarmTrackLength0 : FB_TcAlarm;
END_VAR
// Validate settings
IF THIS^.Length = 0 THEN
	Configure := E_FAIL;
	THIS^.fbFeedback.LastCommandAccepted:= FALSE;	
	IF NOT fbAlarmTrackLength0.bRaised THEN
		fbAlarmTrackLength0.CreateEx(stEventEntry:= TC_EVENTS.CHALET_XPlanar_Events.TrackLength0, bWithConfirmation := FALSE, ipSourceInfo := THIS^.fbSourceInfo);
		fbAlarmTrackLength0.Raise(0);
	END_IF
	RETURN;
ELSE
	fbAlarmTrackLength0.Clear(0,0);	
END_IF



THIS^.eActiveCommand 				:= CHALET_NC.E_NcAxisCommands.Configure;
THIS^.fbFeedback.LastCommandAccepted:= TRUE;		
THIS^.fbFeedback.Busy 				:= TRUE;

THIS^.nSeqConfiguring := 10;
Configure := S_OK;
END_METHOD

METHOD Configuring : HRESULT // This is called until S_OK during system enabling
VAR
	ipEachTrackObj : I_CH_Object;
	nIdx : UDINT;
	ipTrackComObject : ITComObject;
	nParaSize : UDINT;
	pParaData : PVOID;
	hr : HRESULT;
END_VAR
VAR CONSTANT
	N_IDX_OFFSET_PREVIOUS_TRACK 	: UDINT := 16#050300D5; // Parameter(online) in Planar Track object
	N_IDX_OFFSET_SUBSEQUENT_TRACK 	: UDINT := 16#050300D6; // Parameter(online) in Planar Track object	
	N_IDX_OFFSET_IS_CLOSED_LOOP		: UDINT := 16#050300E1; // Parameter(online) in Planar Track object	
END_VAR
Configuring := S_PENDING;
CASE nSeqConfiguring OF
	0: // Idle
		Configuring := S_OK;
		
	10: //Start
		nSeqConfiguring := 200;
		
		
		
	200: //Read information from Track TcCom object
		//Get interface to ComObject
		FW_ObjMgr_GetObjectInstance(oid:= THIS^.OID, iid:= TC_GLOBAL_IID_LIST.IID_ITComObject, pipUnk:= ADR(ipTrackComObject));
	
		IF ipTrackComObject = 0 THEN
			//Error, interface not found
			nSeqConfiguring := nSeqConfiguring + 1000;	
		ELSE
			//Read array of oids PreviousTrackOTCIDs
			nParaSize := SIZEOF(THIS^.PreviousTrackOTCIDs);	pParaData := ADR(THIS^.PreviousTrackOTCIDs);
			hr := ipTrackComObject.TcGetObjPara(pid:=N_IDX_OFFSET_PREVIOUS_TRACK , nData:= nParaSize, pData:= pParaData, pgp:=0 );
			
			//Read array of oids SubsequentTrackOTCIDs
			nParaSize := SIZEOF(THIS^.SubsequentTrackOTCIDs);	pParaData := ADR(THIS^.SubsequentTrackOTCIDs);
			hr := ipTrackComObject.TcGetObjPara(pid:=N_IDX_OFFSET_SUBSEQUENT_TRACK , nData:= nParaSize, pData:= pParaData, pgp:=0 );			
			
			//Read bool CLOSED_LOOP
			nParaSize := SIZEOF(THIS^.bIsClosedLoop);	pParaData := ADR(THIS^.bIsClosedLoop);
			hr := ipTrackComObject.TcGetObjPara(pid:=N_IDX_OFFSET_IS_CLOSED_LOOP , nData:= nParaSize, pData:= pParaData, pgp:=0 );		

			ipTrackComObject.TcRelease();
			nSeqConfiguring := 300;
		END_IF
		
			
	300: // Convert SubsequentTrackOTCIDs to I_XP_Track and add to fbTracksAhead
		fbTracksAhead.Clear();
		FOR nIdx := 0 TO (XPlanarParameterlist.N_MAX_STATIONS_AHEAD_OR_BEHIND-1) DO
			//Get interface to object
			ipEachTrackObj := THIS^.ipXpSystem.Tracks.FindOID(THIS^.SubsequentTrackOTCIDs[nIdx]);
			//convert object -> I_XP_Track. If found, store in list
			IF ToXpTrack(ipEachTrackObj, ipTracksStartFromThis[nIdx]) THEN
				fbTracksAhead.AddObject(ipEachTrackObj);
				
			ELSIF THIS^.SubsequentTrackOTCIDs[nIdx] = 0 THEN
				;//No OTCID
				
			ELSE
				//Error, no track found with following oid
				nSeqConfiguring := nSeqConfiguring + 1000;	
				RETURN;;				
			END_IF
		END_FOR
		nSeqConfiguring := 301;		
	

	301: // Convert PreviousTrackOTCIDs to I_XP_Track and add to fbTracksBehinde
		fbTracksBehinde.Clear();
		FOR nIdx := 0 TO (XPlanarParameterlist.N_MAX_STATIONS_AHEAD_OR_BEHIND-1) DO
			//Get interface to object
			ipEachTrackObj := THIS^.ipXpSystem.Tracks.FindOID(THIS^.PreviousTrackOTCIDs[nIdx]);
			//convert object -> I_XP_Track. If found, store in list
			IF ToXpTrack(ipEachTrackObj, ipTracksEndAtThis[nIdx]) THEN
				fbTracksBehinde.AddObject(ipEachTrackObj);
				
			ELSIF THIS^.PreviousTrackOTCIDs[nIdx] = 0 THEN
				;//No OTCID
				
			ELSE
				//Error, no track found with following oid
				nSeqConfiguring := nSeqConfiguring + 1000;	
				RETURN;;				
			END_IF
		END_FOR			
		nSeqConfiguring := 999;
			
		
	999: // Done
		Configuring := S_OK;
		
	1000..1999://Error
		Configuring := E_FAIL;
END_CASE
END_METHOD

METHOD Disable : HRESULT
VAR_INPUT
END_VAR
IF NOT THIS^.fbFeedback.Busy THEN
	THIS^.eActiveCommand 				:= CHALET_NC.E_NcAxisCommands.Disable;
	THIS^.fbFeedback.LastCommandAccepted:= TRUE;		
	THIS^.fbFeedback.Busy 				:= TRUE;

	THIS^.fbTrack.Disable(fbFeedbackDisable);
	Disable := S_OK;
ELSE
	Disable := S_FALSE;
	THIS^.fbFeedback.LastCommandAccepted:= FALSE;	
END_IF
END_METHOD

METHOD Enable : HRESULT
VAR_INPUT
END_VAR
IF NOT THIS^.fbFeedback.Busy THEN
	THIS^.eActiveCommand 				:= CHALET_NC.E_NcAxisCommands.Enable;
	THIS^.fbFeedback.LastCommandAccepted:= TRUE;		
	THIS^.fbFeedback.Busy 				:= TRUE;

	THIS^.fbTrack.Enable(fbFeedbackEnable);
	Enable := S_OK;
ELSE
	Enable := S_FALSE;
	THIS^.fbFeedback.LastCommandAccepted:= FALSE;	
END_IF
END_METHOD

METHOD AddToGroup : HRESULT
VAR_INPUT
	iGroup : I_XP_Group;
END_VAR
IF NOT THIS^.fbFeedback.Busy THEN
	THIS^.eActiveCommand 				:= CHALET_NC.E_NcAxisCommands.AddToGroupe;
	THIS^.fbFeedback.LastCommandAccepted:= TRUE;		
	THIS^.fbFeedback.Busy 				:= TRUE;
	
	iGroup.AddTrack(THIS^.fbTrack, THIS^.fbFeedbackAddToGrp);
	AddToGroup := S_OK;
ELSE
	AddToGroup := S_FALSE;
	THIS^.fbFeedback.LastCommandAccepted:= FALSE;	
END_IF
END_METHOD

METHOD RemoveFromGroup : HRESULT
IF NOT THIS^.fbFeedback.Busy THEN
	THIS^.eActiveCommand 				:= CHALET_NC.E_NcAxisCommands.RemoveFromGroupe;
	THIS^.fbFeedback.LastCommandAccepted:= TRUE;		
	THIS^.fbFeedback.Busy 				:= TRUE;
	
	THIS^.fbTrack.RemoveFromGroup(THIS^.fbFeedbackRmvFromGrp);
	
	RemoveFromGroup := S_OK;
ELSE
	RemoveFromGroup := S_FALSE;
	THIS^.fbFeedback.LastCommandAccepted:= FALSE;	
END_IF
END_METHOD

METHOD AddMover : HRESULT
VAR_INPUT
	ipMover : I_XP_Mover;
END_VAR
IF ipMover <> 0 THEN
	AddMover := ipMover.JoinTrack(THIS^);
ELSE
	AddMover := E_FAIL;
END_IF
END_METHOD

{attribute 'monitoring':='call'}
PROPERTY ClosedLoop : BOOL
GET
ClosedLoop := bIsClosedLoop;
END_GET
END_PROPERTY

{attribute 'monitoring':='call'}
PROPERTY CtsMoversOnTrack : UINT
GET
THIS^.Prepare();//Prepare a list movers on this track


CtsMoversOnTrack := TO_UINT(THIS^.fbListOfMoversOnTrack.Size);
END_GET
END_PROPERTY

METHOD FB_init : BOOL
VAR_INPUT
	bInitRetains : BOOL; // if TRUE, the retain variables are initialized (warm start / cold start)
	bInCopyCode : BOOL;  // if TRUE, the instance afterwards gets moved into the copy code (online change)
	
	ipSystem : I_CH_Object;
END_VAR
VAR_INST
	{attribute 'hide'}
	bFBInitCalledOnce : BOOL; //Do the following code once during start up and not during onlinechange
END_VAR
//Do the following code once during start up and not during onlinechange
IF NOT bFBInitCalledOnce THEN 
	
	(* Register to the Xplanar System
	   1. Test if the interface exists
	   2. Test if the object implements a "System for Mover" interface 
	*)
	IF ipSystem <> 0 AND_THEN __QUERYINTERFACE(ipSystem,THIS^.ipXpSystem) THEN
		THIS^.ipXpSystem.RegisterTrack(THIS^);
	END_IF
	

END_IF

bFBInitCalledOnce := TRUE;
END_METHOD

{attribute 'monitoring':='call'}
PROPERTY Feedback : I_XP_Feedback
GET
Feedback := THIS^.fbFeedback;
END_GET
END_PROPERTY

(* Calculates which gap the mover should have on a position
	The gap results from the last station crossed.
	If several stations are possible ( switch), the largest gap is displayed here *)
METHOD GapAtPosition : LREAL
VAR_INPUT
	fPosOnTrack : LREAL;//[mm]	
END_VAR
VAR
	ipThisTrack : I_XP_Track := (THIS^);
	bStartAndEndIsOnThisTrack : BOOL;
	ipEachPathOnTrack : I_XP_Path;
END_VAR


THIS^.fbListPathsOnThisTrack.ResetIterator();
WHILE THIS^.fbListPathsOnThisTrack.HasNextObject() DO
	IF __QUERYINTERFACE(THIS^.fbListPathsOnThisTrack.GetNextObject(), ipEachPathOnTrack) THEN
			
		bStartAndEndIsOnThisTrack := ipEachPathOnTrack.StationStart.AccocietedTrack = ipThisTrack AND ipEachPathOnTrack.StationDestination.AccocietedTrack = ipThisTrack; 
			
		//Check if start of route is maybe on this track
		IF (ipEachPathOnTrack.StationStart.AccocietedTrack = ipThisTrack) AND (ipEachPathOnTrack.StationStart.PositionOnTrack > fPosOnTrack) AND NOT bStartAndEndIsOnThisTrack THEN
			//start is after the searched position
			CONTINUE;

		//Check if end of route is maybe on this track
		ELSIF (ipEachPathOnTrack.StationDestination.AccocietedTrack = ipThisTrack) AND (ipEachPathOnTrack.StationDestination.PositionOnTrack <= fPosOnTrack) AND NOT bStartAndEndIsOnThisTrack THEN
			//end is befor the searched position
			CONTINUE;		
			
		//Check if in limit - CLOSED LOOP, SHORT SEGMENT Start > End
		ELSIF F_InLimitTest(fMinimum := ipEachPathOnTrack.StationStart.PositionOnTrack, fInput:= fPosOnTrack, fMaximum := ipEachPathOnTrack.StationDestination.PositionOnTrack) AND bStartAndEndIsOnThisTrack THEN
			//track is outside the searched position
			CONTINUE;		

			
		ELSE
			//The gap is valide, use the largest one
			GapAtPosition := MAX(GapAtPosition, ipEachPathOnTrack.StationStart.MoverGapAtExit);

		END_IF
		
	END_IF
END_WHILE
THIS^.fbListPathsOnThisTrack.RestoreIterator();
END_METHOD

METHOD Initialize : HRESULT
VAR
	hr : HRESULT;
	ipStation : I_XP_Station;
	stVarInfo : __SYSTEM.VAR_INFO;
	pObject : ITComObject;
	sName : STRING;
END_VAR

